(* IEC 61131-3 sources: Lua/, 14 files *)

(* ---- 1#真空脱水.st ---- *)
FUNCTION_BLOCK Dewater
    VAR_STATIC
        // 1#真空脱水控制流--结构体
        TYPE Dewater_1: STRUCT
                bnt_run: BOOL; (* 启动按钮 *)
                bnt_stop: BOOL; (* 停止按钮 *)
                bnt_manual: BOOL; (* 手动按钮 *)
                state: INT; (* 状态 *)
                error_id: INT; (* 错误 *)
                TYPE run: STRUCT
                        todo: BOOL; (* 初始化 *)
                        busy: BOOL; (* 执行中 *)
                        STEP: INT; (* 步数 *)
                        in_time: WORD; (* 计时器输入IN *)
                        skip: BOOL; (* 跳过 *)
                    END_STRUCT
                END_TYPE
                TYPE stop: STRUCT
                        todo: BOOL; (* 初始化 *)
                        busy: BOOL; (* 执行中 *)
                        STEP: INT; (* 步数 *)
                        in_time: WORD; (* 计时器输入IN *)
                        skip: BOOL; (* 跳过 *)
                    END_STRUCT
                END_TYPE
            END_STRUCT
        END_TYPE
        // 1#真空脱水设置时间--结构体
        TYPE Retain_time_D_1 : STRUCT
                preTime : DINT; (* 预处理时间 *)
                openTime_1 : DINT; (* 真空脱水时间 *)
                openTime_2 : DINT; (* 真空脱水时间 *)
                delayTime : DINT; (* 延迟时间 *)
                loopTime : DINT; (* 循环时间 *)
            END_STRUCT
        END_TYPE
        // 1#真空脱水计时器--数组
        Timer_D_1 : ARRAY [0..3] OF TON_TIME;

        CIP_1: "CIP"
        bnt_run: BOOL			启动按钮
        bnt_stop: BOOL			停止按钮
        todo: BOOL			    初始化
        busy: BOOL			    执行中
        step: INT			    步数
        in_time: WORD			计时器输入IN
        error: INT			    错误
        state: INT			    状态

	    Timer_CIP_1	Array[0..10] of TON_TIME

        Retain_time_CIP_1: "CIP_time"
        preTime: DINT
        stepTime_1: DINT
        stepTime_2: DINT
        T102: DINT
        T103: DINT
        T104: DINT
        T105: DINT
        T106: DINT
        T110: DINT
        T107: DINT
        T108: DINT
        T109: DINT
    END_VAR

    /*
        真空脱水一键启动
    */
    // 计时器
    Timer_D_1[0] (IN := #Dewater_1.run.in_time.%X0, PT := #Retain_time_D_1.preTime);
    Timer_D_1[1] (IN := #Dewater_1.run.in_time.%X1, PT := #Retain_time_D_1.openTime_1);

    // 预处理
    IF "Global".Emergency.Dewater_1 THEN
        IF #Dewater_1.bnt_run AND NOT #Dewater_1.run.busy THEN
            "V8016-O" := FALSE;
            "V8021-O" := FALSE;
            "V8011-O" := FALSE;
            "V8026-O" := TRUE;
            #Dewater_1.run.todo := TRUE;
        END_IF;
        IF #Dewater_1.run.todo THEN
            #Dewater_1.state := 1;
            #Dewater_1.run.step := 1;
            #Dewater_1.run.skip := FALSE;
            #Dewater_1.run.in_time := 0;
            #Dewater_1.run.in_time.%X0 := TRUE;
            "ALARM3-O" := TRUE;
            #Dewater_1.bnt_run := FALSE;
        END_IF;
        IF #Dewater_1.run.in_time.%X0 AND #Timer_D_1[0].Q THEN
            #Dewater_1.run.busy := TRUE;
            #Dewater_1.run.todo := FALSE;
            "ALARM3-O" := FALSE;
        ELSE
            #Dewater_1.run.busy := FALSE;
        END_IF;
    ELSE
        #Dewater_1.state := 0;
        #Dewater_1.run.step := 0;
        #Dewater_1.run.in_time := 0;
        #Dewater_1.stop.step := 0;
        #Dewater_1.stop.in_time := 0;
        "ALARM3-O" := FALSE;
    END_IF;

    // 手动时
    IF "Global".Emergency.Dewater_1 AND #Dewater_1.bnt_manual THEN
        #Dewater_1.state := 2;
        #Dewater_1.run.step := 0;
        #Dewater_1.run.in_time := 0;
        #Dewater_1.stop.step := 0;
        #Dewater_1.stop.in_time := 0;
    END_IF;

    // 停止时
    IF "Global".Emergency.Dewater_1 AND #Dewater_1.bnt_stop THEN
        #Dewater_1.state := 3;
        #Dewater_1.run.step := 0;
        #Dewater_1.run.in_time := 0;
    END_IF;

    // 启动中
    IF #Dewater_1.run.busy AND Dewater_1.state = 1 THEN
        // 第1步
        IF #Dewater_1.run.step = 1 THEN
            IF NOT "KV7001-O" THEN
                "KV7001-O" := TRUE;
                #Dewater_1.run.step := 2;
                RETURN;
            END_IF;
            IF "KV7001-O" THEN
                #Dewater_1.run.skip := TRUE;
                #Dewater_1.run.step := 2;
            END_IF;
        END_IF;
        // 第2步
        IF #Dewater_1.run.step = 2 THEN
            IF NOT "A7001-DO" THEN
                IF #Dewater_1.run.skip THEN
                    "A7001-DO" := TRUE;
                    #Dewater_1.run.skip := FALSE;
                    #Dewater_1.run.step := 3;
                    RETURN;
                END_IF;
                #Dewater_1.run.in_time.%X1 := TRUE;
                IF #Dewater_1.run.in_time.%X1 AND #Timer_D_1[1].Q THEN
                    "A7001-DO" := TRUE;
                    #Dewater_1.run.in_time.%X1 := FALSE;
                    #Dewater_1.run.step := 3;
                    RETURN;
                END_IF;
            END_IF;
            IF "A7001-DO" THEN
                #Dewater_1.run.step := 3;
            END_IF;
        END_IF;
        // 第3步
        IF #Dewater_1.run.step = 3 THEN
            IF NOT "F7001-DO" THEN
                IF #Dewater_1.run.skip THEN
                    "F7001-DO" := TRUE;
                    #Dewater_1.run.skip := FALSE;
                    #Dewater_1.run.step := 4;
                    RETURN;
                END_IF;
                #Dewater_1.run.in_time.%X1 := TRUE;
                IF #Dewater_1.run.in_time.%X1 AND #Timer_D_1[1].Q THEN
                    "F7001-DO" := TRUE;
                    #Dewater_1.run.in_time.%X1 := FALSE;
                    #Dewater_1.run.step := 4;
                    RETURN;
                END_IF;
            END_IF;
            IF "F7001-DO" THEN
                #Dewater_1.run.step := 4;
            END_IF;
        END_IF;
        // 第4步
        IF #Dewater_1.run.step = 4 THEN
            IF NOT ( "V8001-O" AND NOT "V8006-O" ) THEN
                IF #Dewater_1.run.skip THEN
                    "V8001-O" := TRUE;
                    "V8006-O" := FALSE;
                    #Dewater_1.run.skip := FALSE;
                    #Dewater_1.run.step := 5;
                    RETURN;
                END_IF;
                #Dewater_1.run.in_time.%X1 := TRUE;
                IF #Dewater_1.run.in_time.%X1 AND #Timer_D_1[1].Q THEN
                    "V8001-O" := TRUE;
                    "V8006-O" := FALSE;
                    #Dewater_1.run.in_time.%X1 := FALSE;
                    #Dewater_1.run.step := 5;
                    RETURN;
                END_IF;
            END_IF;
            IF "V8001-O" AND NOT "V8006-O" THEN
                #Dewater_1.run.step := 5;
            END_IF;
        END_IF;
        // 第5步
        IF #Dewater_1.run.step = 5 THEN
            IF NOT "P8001-DO" THEN
                IF #Dewater_1.run.skip THEN
                    "P8001-DO" := TRUE;
                    #Dewater_1.run.skip := FALSE;
                    #Dewater_1.run.step := 6;
                    RETURN;
                END_IF;
                #Dewater_1.run.in_time.%X1 := TRUE;
                IF #Dewater_1.run.in_time.%X1 AND #Timer_D_1[1].Q THEN
                    "P8001-DO" := TRUE;
                    #Dewater_1.run.in_time.%X1 := FALSE;
                    #Dewater_1.run.step := 6;
                    RETURN;
                END_IF;
            END_IF;
            IF "P8001-DO" THEN
                #Dewater_1.run.step := 6;
            END_IF;
        END_IF;
        // 第6步
        IF #Dewater_1.run.step = 6 THEN
            IF NOT "T7001-DO" THEN
                IF #Dewater_1.run.skip THEN
                    "T7001-DO" := TRUE;
                    #Dewater_1.run.skip := FALSE;
                    #Dewater_1.run.step := 7;
                    RETURN;
                END_IF;
                #Dewater_1.run.in_time.%X1 := TRUE;
                IF #Dewater_1.run.in_time.%X1 AND #Timer_D_1[1].Q THEN
                    "T7001-DO" := TRUE;
                    #Dewater_1.run.in_time.%X1 := FALSE;
                    #Dewater_1.run.step := 7;
                    RETURN;
                END_IF;
            END_IF;
            IF "T7001-DO" THEN
                #Dewater_1.run.step := 7;
            END_IF;
        END_IF;
        // 第7步
        IF #Dewater_1.run.step = 7 THEN
            IF NOT "P7006-DO" THEN
                IF #Dewater_1.run.skip THEN
                    IF "Global".Disp_LIT_7001 > "Global".set_LIT_7001 THEN
                        "P7006-DO" := TRUE;
                        #Dewater_1.run.skip := FALSE;
                        #Dewater_1.run.step := 8;
                        RETURN;
                    ELSE
                        RETURN;
                    END_IF;
                END_IF;
                IF "Global".Disp_LIT_7001 > "Global".set_LIT_7001 THEN
                    #Dewater_1.run.in_time.%X1 := TRUE;
                    IF #Dewater_1.run.in_time.%X1 AND #Timer_D_1[1].Q THEN
                        "P7006-DO" := TRUE;
                        #Dewater_1.run.in_time.%X1 := FALSE;
                        #Dewater_1.run.step := 8;
                        RETURN;
                    END_IF;
                END_IF;
            END_IF;
            IF "P7006-DO" THEN
                #Dewater_1.run.step := 8;
            END_IF;
        END_IF
        // 第8步
        IF #Dewater_1.run.step = 8 THEN
            IF NOT "V7001-O" THEN
                IF #Dewater_1.run.skip THEN
                    "V7001-O" := TRUE;
                    #Dewater_1.run.skip := FALSE;
                    #Dewater_1.run.step := 9;
                    RETURN;
                END_IF;
                #Dewater_1.run.in_time.%X1 := TRUE;
                IF #Dewater_1.run.in_time.%X1 AND #Timer_D_1[1].Q THEN
                    "V7001-O" := TRUE;
                    #Dewater_1.run.in_time.%X1 := FALSE;
                    #Dewater_1.run.step := 9;
                    RETURN;
                END_IF;
            END_IF;
            IF "V7001-O" THEN
                #Dewater_1.run.step := 9;
            END_IF;
        END_IF;
        // 第9步
        IF #Dewater_1.run.step = 9 THEN
            IF NOT "P7001-DO" THEN
                #Dewater_1.run.in_time.%X1 := TRUE;
                IF #Dewater_1.run.in_time.%X1 AND #Timer_D_1[1].Q THEN
                    "P7001-DO" := TRUE;
                    #Dewater_1.run.in_time := 0;
                    #Dewater_1.run.step := 100;
                    RETURN;
                END_IF;
            END_IF;
            IF "P7001-DO" THEN
                #Dewater_1.run.in_time := 0;
                #Dewater_1.run.step := 100;
            END_IF;
        END_IF;
    END_IF;

    /*
        CIP在线清洗
    */
    REGION 计时器
        #Timer_CIP_1[0](IN:=#CIP_1.in_time.%X0, PT:=#Retain_time_CIP_1.preTime);
        #Timer_CIP_1[1](IN := #CIP_1.in_time.%X1, PT := #Retain_time_CIP_1.stepTime_1);
        #Timer_CIP_1[2](IN := #CIP_1.in_time.%X2, PT := #Retain_time_CIP_1.T102);
        #Timer_CIP_1[3](IN := #CIP_1.in_time.%X3, PT := #Retain_time_CIP_1.T103);
        #Timer_CIP_1[4](IN := #CIP_1.in_time.%X4, PT := #Retain_time_CIP_1.T104);
        #Timer_CIP_1[5](IN := #CIP_1.in_time.%X5, PT := #Retain_time_CIP_1.T105);
        #Timer_CIP_1[6](IN := #CIP_1.in_time.%X6, PT := #Retain_time_CIP_1.T106);
        #Timer_CIP_1[7](IN := #CIP_1.in_time.%X7, PT := #Retain_time_CIP_1.T107);
        #Timer_CIP_1[8](IN := #CIP_1.in_time.%X8, PT := #Retain_time_CIP_1.T108);
        #Timer_CIP_1[9](IN := #CIP_1.in_time.%X9, PT := #Retain_time_CIP_1.T109);
        #Timer_CIP_1[10](IN := #CIP_1.in_time.%X10, PT := #Retain_time_CIP_1.T110);
    END_REGION

    REGION 预处理
        // 初始化
        IF "Global".Emergency.Dewater_1 THEN
            IF #Dewater_1.state = 1 AND #Dewater_1.run.step = 100 AND #CIP_1.bnt_run AND NOT #CIP_1.busy THEN
                #CIP_1.todo := TRUE;
            END_IF;
            IF #CIP_1.todo THEN
                #CIP_1.state := 1;
                #CIP_1.step := 1;
                #CIP_1.in_time := 0;
                #CIP_1.in_time.%X0 := TRUE;
                #CIP_1.bnt_run := FALSE;
                #CIP_1.todo := FALSE;
            END_IF;
            IF #CIP_1.in_time.%X0 AND #Timer_CIP_1[0].Q THEN
                #CIP_1.busy := TRUE;
            ELSE
                #CIP_1.busy := FALSE;
            END_IF;
        ELSE
            #CIP_1.state := 0;
            #CIP_1.step := 0;
            #CIP_1.in_time := 0;
        END_IF;
    END_REGION

    REGION CIP运行中
        IF #CIP_1.busy AND #CIP_1.state = 1 THEN
            // step 1
            IF #CIP_1.step = 1 THEN
                "V8006-O" := TRUE;
                #CIP_1.step := 2;
            END_IF;
            // step 2
            IF #CIP_1.step = 2 THEN
                #CIP_1.in_time.%X2 := TRUE;
                IF #CIP_1.in_time.%X2 AND #Timer_CIP_1[2].Q THEN
                    "V8001-O" := FALSE;
                    #CIP_1.in_time.%X2:= FALSE;
                    #CIP_1.step := 3;
                END_IF;
            END_IF;
            // step 3
            IF #CIP_1.step = 3 THEN
                #CIP_1.in_time.%X3 := TRUE;
                IF #CIP_1.in_time.%X3 AND #Timer_CIP_1[3].Q THEN
                    "P8001-DO" := FALSE;
                    "Global".PID_7101.Man_enable := TRUE;
                    "Global".PID_7101.Man_value := 0;
                    "V8006-O" := FALSE;
                    "V8011-O" := TRUE;
                    #CIP_1.in_time.%X3 := FALSE;
                    #CIP_1.step := 4;
                END_IF;
            END_IF;
            // step 4
            IF #CIP_1.step = 4 THEN
                #CIP_1.in_time.%X4 := TRUE;
                IF #CIP_1.in_time.%X4 AND #Timer_CIP_1[4].Q THEN
                    "V8011-O" := FALSE;
                    #CIP_1.in_time.%X4 := FALSE;
                    #CIP_1.step := 5;
                END_IF;
            END_IF;
            // step 5
            IF #CIP_1.step = 5 THEN
                #CIP_1.in_time.%X1 := TRUE;
                IF #CIP_1.in_time.%X1 AND #Timer_CIP_1[1].Q THEN
                    "KV7001-O" := FALSE;
                    #CIP_1.in_time.%X1 := FALSE;
                    #CIP_1.step := 6;
                    RETURN;
                END_IF;
            END_IF;
            // step 6
            IF #CIP_1.step = 6 THEN
                #CIP_1.in_time.%X1 := TRUE;
                IF #CIP_1.in_time.%X1 AND #Timer_CIP_1[1].Q THEN
                    "P7001-DO" := FALSE;
                    "V7001-O" := FALSE;
                    #CIP_1.in_time.%X1 := FALSE;
                    #CIP_1.step := 7;
                    RETURN;
                END_IF;
            END_IF;
            // step 7
            IF #CIP_1.step = 7 THEN
                #CIP_1.in_time.%X1 := TRUE;
                IF #CIP_1.in_time.%X1 AND #Timer_CIP_1[1].Q THEN
                    "P7006-DO" := FALSE;
                    #CIP_1.in_time.%X1 := FALSE;
                    #CIP_1.step := 8;
                    RETURN;
                END_IF;
            END_IF;
            // step 8
            IF #CIP_1.step = 8 THEN
                #CIP_1.in_time.%X1 := TRUE;
                IF #CIP_1.in_time.%X1 AND #Timer_CIP_1[1].Q THEN
                    "T7001-DO" := FALSE;
                    #CIP_1.in_time.%X1 := FALSE;
                    #CIP_1.step := 9;
                    RETURN;
                END_IF;
            END_IF;
            // step 9
            IF #CIP_1.step = 9 THEN
                #CIP_1.in_time.%X1 := TRUE;
                IF #CIP_1.in_time.%X1 AND #Timer_CIP_1[1].Q THEN
                    "V8016-O" := TRUE;
                    "V8017-O" := FALSE;
                    "V8018-O" := FALSE;
                    "V8019-O" := FALSE;
                    "V8020-O" := FALSE;
                    "V8021-O" := FALSE;
                    #CIP_1.in_time.%X1 := FALSE;
                    #CIP_1.step := 901;
                    RETURN;
                END_IF;
            END_IF;
            // step 901
            IF #CIP_1.step = 901 THEN
                #CIP_1.in_time.%X1 := TRUE;
                IF #CIP_1.in_time.%X1 AND #Timer_CIP_1[1].Q THEN
                    "P8007-DO" := TRUE;
                    #CIP_1.in_time.%X1 := FALSE;
                    #CIP_1.step := 10;
                    RETURN;
                END_IF;
            END_IF;
            // step 10
            IF #CIP_1.step = 10 THEN
                #CIP_1.in_time.%X5 := TRUE;
                IF #CIP_1.in_time.%X5 AND #Timer_CIP_1[5].Q THEN
                    "P8007-DO" := FALSE;
                    "V8016-O" := FALSE;
                    #CIP_1.in_time.%X5 := FALSE;
                    #CIP_1.step := 11;
                END_IF;
            END_IF;
            // step 11
            IF #CIP_1.step = 11 THEN
                #CIP_1.in_time.%X6 := TRUE;
                IF #CIP_1.in_time.%X6 AND #Timer_CIP_1[6].Q THEN
                    "V8026-O" := TRUE;
                    "V8032-O" := TRUE;
                    #CIP_1.in_time.%X6 := FALSE;
                    #CIP_1.step := 12;
                END_IF;
            END_IF;
            // step 12
            IF #CIP_1.step = 12 THEN
                #CIP_1.in_time.%X10 := TRUE;
                IF #CIP_1.in_time.%X10 AND #Timer_CIP_1[10].Q THEN
                    "V8032-O" := FALSE;
                    "Global".set_Hz_F7001 := 10.0;
                    #CIP_1.in_time.%X10 := FALSE;
                    #CIP_1.step := 13;
                END_IF;
            END_IF;
            // step 13
            IF #CIP_1.step = 13 THEN
                #CIP_1.in_time.%X1 := TRUE;
                IF #CIP_1.in_time.%X1 AND #Timer_CIP_1[1].Q THEN
                    "V8016-O" := TRUE;
                    "V8017-O" := FALSE;
                    "V8018-O" := FALSE;
                    "V8019-O" := FALSE;
                    "V8020-O" := FALSE;
                    "V8021-O" := FALSE;
                    #CIP_1.in_time.%X1 := FALSE;
                    #CIP_1.step := 1301;
                    RETURN;
                END_IF;
            END_IF;
            // step 1301
            IF #CIP_1.step = 1301 THEN
                #CIP_1.in_time.%X1 := TRUE;
                IF #CIP_1.in_time.%X1 AND #Timer_CIP_1[1].Q THEN
                    "P8007-DO" := TRUE;
                    #CIP_1.in_time.%X1 := FALSE;
                    #CIP_1.step := 14;
                    RETURN;
                END_IF;
            END_IF;
            // step 14
            IF #CIP_1.step = 14 THEN
                #CIP_1.in_time.%X7 := TRUE;
                IF #CIP_1.in_time.%X7 AND #Timer_CIP_1[7].Q THEN
                    "P8007-DO" := FALSE;
                    "V8016-O" := FALSE;
                    #CIP_1.in_time.%X7 := FALSE;
                    #CIP_1.step := 15;
                END_IF;
            END_IF;
            // step 15
            IF #CIP_1.step = 15 THEN
                #CIP_1.in_time.%X8 := TRUE;
                IF #CIP_1.in_time.%X8 AND #Timer_CIP_1[8].Q THEN
                    "V8026-O" := FALSE;
                    "V8031-O" := TRUE;
                    #CIP_1.in_time.%X8 := FALSE;
                    #CIP_1.step := 16;
                END_IF;
            END_IF;
            // step 16
            IF #CIP_1.step = 16 THEN
                #CIP_1.in_time.%X9 := TRUE;
                IF #CIP_1.in_time.%X9 AND #Timer_CIP_1[9].Q THEN
                    "V8031-O" := FALSE;
                    #CIP_1.in_time.%X9 := FALSE;
                    #CIP_1.step := 17;
                END_IF;
            END_IF;
            // step 17
            IF #CIP_1.step = 17 THEN
                #CIP_1.in_time.%X1 := TRUE;
                IF #CIP_1.in_time.%X1 AND #Timer_CIP_1[1].Q THEN
                    "A7001-DO" := FALSE;
                    #CIP_1.in_time.%X1 := FALSE;
                    #CIP_1.step := 18;
                    RETURN;
                END_IF;
            END_IF;
            // step 18
            IF #CIP_1.step = 18 THEN
                #CIP_1.in_time.%X1 := TRUE;
                IF #CIP_1.in_time.%X1 AND #Timer_CIP_1[1].Q THEN
                    "F7001-DO" := FALSE;
                    #CIP_1.in_time.%X1 := FALSE;
                    #CIP_1.step := 19;
                END_IF;
            END_IF;
        END_IF;
    END_REGION
END_FUNCTION_BLOCK

(* ---- 真空脱水_3_25.st ---- *)
FUNCTION_BLOCK Dewater
    VAR_STAT
        // 1#真空脱水控制流--结构体
        TYPE Dewater_1: STRUCT
                bnt_run: BOOL; (* 启动按钮 *)
                bnt_stop: BOOL; (* 停止按钮 *)
                bnt_manual: BOOL; (* 手动按钮 *)
                state: INT; (* 状态 *)
                TYPE run: STRUCT
                        todo: BOOL; (* 初始化 *)
                        busy: BOOL; (* 执行中 *)
                        STEP: INT; (* 步数 *)
                        in_time: WORD; (* 计时器输入IN *)
                        skip: BOOL; (* 跳过 *)
                    END_STRUCT
                END_TYPE
                TYPE stop: STRUCT
                        todo: BOOL; (* 初始化 *)
                        busy: BOOL; (* 执行中 *)
                        STEP: INT; (* 步数 *)
                        in_time: WORD; (* 计时器输入IN *)
                        skip: BOOL; (* 跳过 *)
                    END_STRUCT
                END_TYPE
            END_STRUCT
        END_TYPE
        // 1#真空脱水设置时间--结构体
        TYPE Retain_time_D_1 : STRUCT
                preTime : DINT; (* 预处理时间 *)
                openTime_1 : DINT; (* 真空脱水时间 *)
                openTime_2 : DINT; (* 真空脱水时间 *)
                delayTime : DINT; (* 延迟时间 *)
                loopTime : DINT; (* 循环时间 *)
            END_STRUCT
        END_TYPE
        // 1#真空脱水计时器--数组
        Timer_D_1 : ARRAY [0..3] OF TON_TIME;
    END_VAR

    // 计时器
    Timer_D_1[0](IN := #Dewater_1.run.in_time.%X0, PT := #Retain_time_D_1.preTime);
    Timer_D_1[1](IN := #Dewater_1.run.in_time.%X0, PT := #Retain_time_D_1.openTime_1);

    // 预处理
    IF "Global".Emergency.Dewater_1 THEN
    IF #Dewater_1.bnt_run AND NOT #Dewater_1.run.busy THEN
        #Dewater_1.run.todo := TRUE;
    END_IF;
    IF #Dewater_1.run.todo THEN
        #Dewater_1.state := 1;
        #Dewater_1.run.step := 1;
        #Dewater_1.run.skip := FALSE;
        #Dewater_1.run.in_time := 0;
        #Dewater_1.run.in_time.%X0 := TRUE;
        "ALARM1-O" := TRUE;
        #Dewater_1.bnt_run := FALSE;
        #Dewater_1.run.todo := FALSE;
    END_IF;

    END_IF;

END_FUNCTION_BLOCK

(* ---- 顺序启动_最新.st ---- *)
FUNCTION_BLOCK Extraction
    VAR_GLOBAL
        //提取单元自动启动关键属性--结构体
        TYPE Common_M_1_run : STRUCT
                bnt_run : BOOL; (* 自动启动 *)
                bnt_stop : BOOL; (* 自动停止 *)
                todo : BOOL; (* 是否跳过步骤1 *)
                busy : BOOL; (* 自动正在执行 *)
                step : INT; (* 自动运行步骤 *)
                in_time : WORD; (* 控制计时器输入IN通断 *)
                manual_enable : BOOL; (* 手动模式按钮 *)
                state : INT; (* 提取单元状态都在此处显示 *)
            END_STRUCT
        END_TYPE

        //提取单元自动启动设定时间--结构体
        TYPE Retain_M5000_run : STRUCT
                preTime : DINT; (* 自动启动预处理时间 *)
                openTime_1 : DINT; (* 自动启动电机延时打开时间 *)
            END_STRUCT
        END_TYPE

        //提取单元启动--通电延时计时器
        Timer_M5000_run : ARRAY[0..2] of TON_TIME;
        (*
            Timer_M5000_run[0]......预处理--计时器
            Timer_M5000_run[1]......电机打开延时--计时器
        *)
    END_VAR

    /* *
    **计时器
    */
    #Timer_M5000_run[0](IN := #Common_M_1_run.in_time.%X0, PT := #Retain_M5000_run.preTime);
    #Timer_M5000_run[1](IN := #Common_M_1_run.in_time.%X1, PT := #Retain_M5000_run.openTime_1);

    /* *
    **预处理
    */
    IF "Global".Emergency.Extraction_1 AND #Common_M_1_run.bnt_run AND NOT #Common_M_1_run.busy THEN
    #Common_M_1_run.state := 1;
    #Common_M_1_run.step := 1;
    #Common_M_1_run.in_time := 0;
    #Common_M_1_run.todo := FALSE;
    #Common_M_1_run.in_time.%X0 := TRUE;
    END_IF;
    IF #Common_M_1_run.in_time.%X0 AND #Timer_M5000_run[0].Q THEN
    #Common_M_1_run.bnt_run := FALSE;
    #Common_M_1_run.busy := TRUE;
    ELSE
    #Common_M_1_run.busy := FALSE;
    END_IF;

    //急停时
    IF NOT "Global".Emergency.Extraction_1 THEN
    #Common_M_1_run.state := 0;
    #Common_M_1_run.step := 0;
    #Common_M_1_run.in_time := 0;
    #Common_M_1_run.bnt_run := FALSE;
    END_IF;

    //手动时
    IF "Global".Emergency.Extraction_1 AND #Common_M_1_run.manual_enable THEN
    #Common_M_1_run.state := 2;
    #Common_M_1_run.step := 0;
    #Common_M_1_run.in_time := 0;
    #Common_M_1_run.bnt_run := FALSE;
    END_IF;

    //停止时
    IF "Global".Emergency.Extraction_1 AND #Common_M_1_run.bnt_stop THEN
    #Common_M_1_run.step := 0;
    #Common_M_1_run.in_time := 0;
    #Common_M_1_run.bnt_run := FALSE;
    END_IF;

    /* *
    **运行时
    */
    IF #Common_M_1_run.busy AND #Common_M_1_run.state = 1 THEN
    //step1
    IF #Common_M_1_run.step = 1 THEN
        IF NOT "M5203-DO" THEN
            "M5203-DO" := TRUE;
            #Common_M_1_run.step := 2;
            RETURN;
        END_IF;
        IF "M5203-DO" THEN
            #Common_M_1_run.todo := TRUE;
            #Common_M_1_run.step := 2;
        END_IF;
    END_IF;
    //step2
    IF #Common_M_1_run.step = 2 THEN
        IF NOT "M5103-DO" THEN
            IF #Common_M_1_run.todo THEN
                "M5103-DO" := TRUE;
                #Common_M_1_run.todo := FALSE;
                #Common_M_1_run.step := 3;
                RETURN;
            END_IF;
            #Common_M_1_run.in_time.%X1 := TRUE;
            IF #Common_M_1_run.in_time.%X1 AND #Timer_M5000_run[1].Q THEN
                "M5103-DO" := TRUE;
                #Common_M_1_run.in_time.%X1 := FALSE;
                #Common_M_1_run.step := 3;
                RETURN;
            END_IF;
        END_IF;
        IF "M5103-DO" THEN
            #Common_M_1_run.step := 3;
        END_IF;
    END_IF;
    //step3
    IF #Common_M_1_run.step = 3 THEN
        IF NOT "M5202-DO" THEN
            IF #Common_M_1_run.todo THEN
                "M5202-DO" := TRUE;
                #Common_M_1_run.todo := FALSE;
                #Common_M_1_run.step := 4;
                RETURN;
            END_IF;
            #Common_M_1_run.in_time.%X1 := TRUE;
            IF #Common_M_1_run.in_time.%X1 AND #Timer_M5000_run[1].Q THEN
                "M5202-DO" := TRUE;
                #Common_M_1_run.in_time.%X1 := FALSE;
                #Common_M_1_run.step := 4;
                RETURN;
            END_IF;
        END_IF;
        IF "M5202-DO" THEN
            #Common_M_1_run.step := 4;
        END_IF;
    END_IF;
    //step4
    IF #Common_M_1_run.step = 4 THEN
        IF NOT "M5102-DO" THEN
            IF #Common_M_1_run.todo THEN
                "M5102-DO" := TRUE;
                #Common_M_1_run.todo := FALSE;
                #Common_M_1_run.step := 5;
                RETURN;
            END_IF;
            #Common_M_1_run.in_time.%X1 := TRUE;
            IF #Common_M_1_run.in_time.%X1 AND #Timer_M5000_run[1].Q THEN
                "M5102-DO" := TRUE;
                #Common_M_1_run.in_time.%X1 := FALSE;
                #Common_M_1_run.step := 5;
                RETURN;
            END_IF;
        END_IF;
        IF "M5102-DO" THEN
            #Common_M_1_run.step := 5;
        END_IF;
    END_IF;
    //step5
    IF #Common_M_1_run.step = 5 THEN
        IF NOT "M5401-DO" THEN
            IF #Common_M_1_run.todo THEN
                "M5401-DO" := TRUE;
                #Common_M_1_run.todo := FALSE;
                #Common_M_1_run.step := 6;
                RETURN;
            END_IF;
            #Common_M_1_run.in_time.%X1 := TRUE;
            IF #Common_M_1_run.in_time.%X1 AND #Timer_M5000_run[1].Q THEN
                "M5401-DO" := TRUE;
                #Common_M_1_run.in_time.%X1 := FALSE;
                #Common_M_1_run.step := 6;
                RETURN;
            END_IF;
        END_IF;
        IF "M5401-DO" THEN
            #Common_M_1_run.step := 6;
        END_IF;
    END_IF;
    //step6
    IF #Common_M_1_run.step = 6 THEN
        IF NOT "M5301-DO" THEN
            IF #Common_M_1_run.todo THEN
                "M5301-DO" := TRUE;
                #Common_M_1_run.todo := FALSE;
                #Common_M_1_run.step := 7;
                RETURN;
            END_IF;
            #Common_M_1_run.in_time.%X1 := TRUE;
            IF #Common_M_1_run.in_time.%X1 AND #Timer_M5000_run[1].Q THEN
                "M5301-DO" := TRUE;
                #Common_M_1_run.in_time.%X1 := FALSE;
                #Common_M_1_run.step := 7;
                RETURN;
            END_IF;
        END_IF;
        IF "M5301-DO" THEN
            #Common_M_1_run.step := 7;
        END_IF;
    END_IF;
    //step7
    IF #Common_M_1_run.step = 7 THEN
        IF NOT "M5201-DO" THEN
            IF #Common_M_1_run.todo THEN
                "M5201-DO" := TRUE;
                #Common_M_1_run.todo := FALSE;
                #Common_M_1_run.step := 8;
                RETURN;
            END_IF;
            #Common_M_1_run.in_time.%X1 := TRUE;
            IF #Common_M_1_run.in_time.%X1 AND #Timer_M5000_run[1].Q THEN
                "M5201-DO" := TRUE;
                #Common_M_1_run.in_time.%X1 := FALSE;
                #Common_M_1_run.step := 8;
                RETURN;
            END_IF;
        END_IF;
        IF "M5201-DO" THEN
            #Common_M_1_run.step := 8;
        END_IF;
    END_IF;
    //step8
    IF #Common_M_1_run.step = 8 THEN
        IF NOT "M5101-DO" THEN
            IF #Common_M_1_run.todo THEN
                "M5101-DO" := TRUE;
                #Common_M_1_run.todo := FALSE;
                #Common_M_1_run.step := 9;
                RETURN;
            END_IF;
            #Common_M_1_run.in_time.%X1 := TRUE;
            IF #Common_M_1_run.in_time.%X1 AND #Timer_M5000_run[1].Q THEN
                "M5101-DO" := TRUE;
                #Common_M_1_run.in_time.%X1 := FALSE;
                #Common_M_1_run.step := 9;
                RETURN;
            END_IF;
        END_IF;
        IF "M5101-DO" THEN
            #Common_M_1_run.step := 9;
        END_IF;
    END_IF;
    //step9
    IF #Common_M_1_run.step = 9 THEN
        IF NOT "P5005-DO" THEN
            IF #Common_M_1_run.todo THEN
                "P5005-DO" := TRUE;
                #Common_M_1_run.todo := FALSE;
                #Common_M_1_run.step := 10;
                RETURN;
            END_IF;
            #Common_M_1_run.in_time.%X1 := TRUE;
            IF #Common_M_1_run.in_time.%X1 AND #Timer_M5000_run[1].Q THEN
                "P5005-DO" := TRUE;
                #Common_M_1_run.in_time.%X1 := FALSE;
                #Common_M_1_run.step := 10;
                RETURN;
            END_IF;
        END_IF;
        IF "P5005-DO" THEN
            #Common_M_1_run.step := 10;
        END_IF;
    END_IF;
    //step10
    IF #Common_M_1_run.step = 10 THEN
        IF NOT "P5003-DO" THEN
            IF #Common_M_1_run.todo THEN
                "P5003-DO" := TRUE;
                #Common_M_1_run.todo := FALSE;
                #Common_M_1_run.step := 11;
                RETURN;
            END_IF;
            #Common_M_1_run.in_time.%X1 := TRUE;
            IF #Common_M_1_run.in_time.%X1 AND #Timer_M5000_run[1].Q THEN
                "P5003-DO" := TRUE;
                #Common_M_1_run.in_time.%X1 := FALSE;
                #Common_M_1_run.step := 11;
                RETURN;
            END_IF;
        END_IF;
        IF "P5003-DO" THEN
            #Common_M_1_run.step := 11;
        END_IF;
    END_IF;
    //step11
    IF #Common_M_1_run.step = 11 THEN
        IF NOT "P5201-DO" THEN
            IF #Common_M_1_run.todo THEN
                "P5201-DO" := TRUE;
                #Common_M_1_run.todo := FALSE;
                #Common_M_1_run.step := 12;
                RETURN;
            END_IF;
            #Common_M_1_run.in_time.%X1 := TRUE;
            IF #Common_M_1_run.in_time.%X1 AND #Timer_M5000_run[1].Q THEN
                "P5201-DO" := TRUE;
                #Common_M_1_run.in_time.%X1 := FALSE;
                #Common_M_1_run.step := 12;
                RETURN;
            END_IF;
        END_IF;
        IF "P5201-DO" THEN
            #Common_M_1_run.step := 12;
        END_IF;
    END_IF;
    //step12
    IF #Common_M_1_run.step = 12 THEN
        IF NOT "P5101-DO" THEN
            IF #Common_M_1_run.todo THEN
                "P5101-DO" := TRUE;
                #Common_M_1_run.todo := FALSE;
                #Common_M_1_run.step := 13;
                RETURN;
            END_IF;
            #Common_M_1_run.in_time.%X1 := TRUE;
            IF #Common_M_1_run.in_time.%X1 AND #Timer_M5000_run[1].Q THEN
                "P5101-DO" := TRUE;
                #Common_M_1_run.in_time.%X1 := FALSE;
                #Common_M_1_run.step := 13;
                RETURN;
            END_IF;
        END_IF;
        IF "P5101-DO" THEN
            #Common_M_1_run.step := 13;
        END_IF;
    END_IF;
    //step13
    IF #Common_M_1_run.step = 13 THEN
        IF NOT "P5206-DO" THEN
            IF #Common_M_1_run.todo THEN
                "P5206-DO" := TRUE;
                #Common_M_1_run.todo := FALSE;
                #Common_M_1_run.step := 14;
                RETURN;
            END_IF;
            #Common_M_1_run.in_time.%X1 := TRUE;
            IF #Common_M_1_run.in_time.%X1 AND #Timer_M5000_run[1].Q THEN
                "P5206-DO" := TRUE;
                #Common_M_1_run.in_time.%X1 := FALSE;
                #Common_M_1_run.step := 14;
                RETURN;
            END_IF;
        END_IF;
        IF "P5206-DO" THEN
            #Common_M_1_run.step := 14;
        END_IF;
    END_IF;
    //step14
    IF #Common_M_1_run.step = 14 THEN
        IF NOT "P5106-DO" THEN
            IF #Common_M_1_run.todo THEN
                "P5106-DO" := TRUE;
                #Common_M_1_run.todo := FALSE;
                #Common_M_1_run.step := 15;
                RETURN;
            END_IF;
            #Common_M_1_run.in_time.%X1 := TRUE;
            IF #Common_M_1_run.in_time.%X1 AND #Timer_M5000_run[1].Q THEN
                "P5106-DO" := TRUE;
                #Common_M_1_run.in_time.%X1 := FALSE;
                #Common_M_1_run.step := 15;
                RETURN;
            END_IF;
        END_IF;
        IF "P5106-DO" THEN
            #Common_M_1_run.step := 15;
        END_IF;
    END_IF;
    //step15
    IF #Common_M_1_run.step = 15 THEN
        IF NOT "P5204-DO" THEN
            IF #Common_M_1_run.todo THEN
                "P5204-DO" := TRUE;
                #Common_M_1_run.todo := FALSE;
                #Common_M_1_run.step := 16;
                RETURN;
            END_IF;
            #Common_M_1_run.in_time.%X1 := TRUE;
            IF #Common_M_1_run.in_time.%X1 AND #Timer_M5000_run[1].Q THEN
                "P5204-DO" := TRUE;
                #Common_M_1_run.in_time.%X1 := FALSE;
                #Common_M_1_run.step := 16;
                RETURN;
            END_IF;
        END_IF;
        IF "P5204-DO" THEN
            #Common_M_1_run.step := 16;
        END_IF;
    END_IF;
    //step16
    IF #Common_M_1_run.step = 16 THEN
        IF NOT "P5104-DO" THEN
            IF #Common_M_1_run.todo THEN
                "P5104-DO" := TRUE;
                #Common_M_1_run.todo := FALSE;
                #Common_M_1_run.step := 17;
                RETURN;
            END_IF;
            #Common_M_1_run.in_time.%X1 := TRUE;
            IF #Common_M_1_run.in_time.%X1 AND #Timer_M5000_run[1].Q THEN
                "P5104-DO" := TRUE;
                #Common_M_1_run.in_time.%X1 := FALSE;
                #Common_M_1_run.step := 17;
                RETURN;
            END_IF;
        END_IF;
        IF "P5104-DO" THEN
            #Common_M_1_run.step := 17;
        END_IF;
    END_IF;
    //step17
    IF #Common_M_1_run.step = 17 THEN
        IF NOT "P5402-DO" THEN
            IF #Common_M_1_run.todo THEN
                "P5402-DO" := TRUE;
                #Common_M_1_run.todo := FALSE;
                #Common_M_1_run.step := 18;
                RETURN;
            END_IF;
            #Common_M_1_run.in_time.%X1 := TRUE;
            IF #Common_M_1_run.in_time.%X1 AND #Timer_M5000_run[1].Q THEN
                "P5402-DO" := TRUE;
                #Common_M_1_run.in_time.%X1 := FALSE;
                #Common_M_1_run.step := 18;
                RETURN;
            END_IF;
        END_IF;
        IF "P5402-DO" THEN
            #Common_M_1_run.step := 18;
        END_IF;
    END_IF;
    //step18
    IF #Common_M_1_run.step = 18 THEN
        IF NOT "P5302-DO" THEN
            IF #Common_M_1_run.todo THEN
                "P5302-DO" := TRUE;
                #Common_M_1_run.todo := FALSE;
                #Common_M_1_run.step := 19;
                RETURN;
            END_IF;
            #Common_M_1_run.in_time.%X1 := TRUE;
            IF #Common_M_1_run.in_time.%X1 AND #Timer_M5000_run[1].Q THEN
                "P5302-DO" := TRUE;
                #Common_M_1_run.in_time.%X1 := FALSE;
                #Common_M_1_run.step := 19;
                RETURN;
            END_IF;
        END_IF;
        IF "P5302-DO" THEN
            #Common_M_1_run.step := 19;
        END_IF;
    END_IF;
    //step19
    IF #Common_M_1_run.step = 19 THEN
        IF NOT "P5202-DO" THEN
            IF #Common_M_1_run.todo THEN
                "P5202-DO" := TRUE;
                #Common_M_1_run.todo := FALSE;
                #Common_M_1_run.step := 20;
                RETURN;
            END_IF;
            #Common_M_1_run.in_time.%X1 := TRUE;
            IF #Common_M_1_run.in_time.%X1 AND #Timer_M5000_run[1].Q THEN
                "P5202-DO" := TRUE;
                #Common_M_1_run.in_time.%X1 := FALSE;
                #Common_M_1_run.step := 20;
                RETURN;
            END_IF;
        END_IF;
        IF "P5202-DO" THEN
            #Common_M_1_run.step := 20;
        END_IF;
    END_IF;
    //step20
    IF #Common_M_1_run.step = 20 THEN
        IF NOT "P5102-DO" THEN
            IF #Common_M_1_run.todo THEN
                "P5102-DO" := TRUE;
                #Common_M_1_run.todo := FALSE;
                #Common_M_1_run.in_time := 0;
                #Common_M_1_run.step := 100;
                RETURN;
            END_IF;
            #Common_M_1_run.in_time.%X1 := TRUE;
            IF #Common_M_1_run.in_time.%X1 AND #Timer_M5000_run[1].Q THEN
                "P5102-DO" := TRUE;
                #Common_M_1_run.in_time := 0;
                #Common_M_1_run.step := 100;
                RETURN;
            END_IF;
        END_IF;
        IF "P5102-DO" THEN
            #Common_M_1_run.in_time := 0;
            #Common_M_1_run.step := 100;
        END_IF;
    END_IF;
    END_IF;
END_FUNCTION_BLOCK

(* ---- 11_15项目离心筛组控制程序修改.st ---- *)
REGION 预处理
    #"Motor-Runtimer"[0]( IN := #"Comm-run".busy, PT := #"Screen-Time"."PT-pretime-m");
    #"Motor-Runtimer"[1]( IN := #"Comm-run"."in-timer".%X1, PT := #"Screen-Time"."PT-runtime");
    #"Motor-Runtimer"[2]( IN := #"Comm-run"."in-timer".%X2, PT := #"Screen-Time"."PT-runtime");

    IF "Debug".Unit_estop_state[2] AND #bnt_manual THEN
        "Debug".Screen_state := 2;
        "Manual".M5101.man_enable := TRUE;
        "Manual".M5201.man_enable := TRUE;
        "Manual".M5002.man_enable := TRUE;
        "Manual".M5003.man_enable := TRUE;
        "Manual".M5004.man_enable := TRUE;
        "Manual".P5101.man_enable := TRUE;
        "Manual".P5102.man_enable := TRUE;
        "Manual".P5201.man_enable := TRUE;
        "Manual".P5202.man_enable := TRUE;
        "Manual".P5003.man_enable := TRUE;
        "Manual".P5004.man_enable := TRUE;
        "Manual".P5005.man_enable := TRUE;
        "Manual".P5006.man_enable := TRUE;
        "Manual".P5007.man_enable := TRUE;
        "Manual".P5008.man_enable := TRUE;
        "Manual".P5009.man_enable := TRUE;
        "Manual".P5010.man_enable := TRUE;
    END_IF;

    IF "Debug".Unit_estop_state[2] AND #bnt_auto THEN
        "Debug".Screen_state := 1;
        "Manual".M5101.man_enable := FALSE;
        "Manual".M5201.man_enable := FALSE;
        "Manual".M5002.man_enable := FALSE;
        "Manual".M5003.man_enable := FALSE;
        "Manual".M5004.man_enable := FALSE;
        "Manual".P5101.man_enable := FALSE;
        "Manual".P5102.man_enable := FALSE;
        "Manual".P5201.man_enable := FALSE;
        "Manual".P5202.man_enable := FALSE;
        "Manual".P5003.man_enable := FALSE;
        "Manual".P5004.man_enable := FALSE;
        "Manual".P5005.man_enable := FALSE;
        "Manual".P5006.man_enable := FALSE;
        "Manual".P5007.man_enable := FALSE;
        "Manual".P5008.man_enable := FALSE;
        "Manual".P5009.man_enable := FALSE;
        "Manual".P5010.man_enable := FALSE;
    END_IF;

    IF "Debug".Unit_estop_state[2] AND "Debug".Screen_state = 1 THEN
        IF #"Comm-run"."bnt-run" AND NOT #"Comm-run".busy THEN
            #"Comm-run".todo := 1;
            //复位工艺停止
            #"Comm-stop"."in-timer" := 0;
            #"Comm-stop".todo := 0;
            #"Comm-stop".busy := 0;
            #"Comm-stop".done := 0;
            #"Comm-stop".step := 0;
        END_IF;
        IF #"Comm-run".todo THEN
            #"Comm-run".busy := 1;
            #"Comm-run".step := 1;
            #"Comm-run".todo := 0;
        END_IF;
    ELSE
        #"Comm-run"."in-timer" := 0;
        #"Comm-run".todo := 0;
        #"Comm-run".busy := 0;
        #"Comm-run".done := 0;
        #"Comm-run".step := 0;
    END_IF;
END_REGION

REGION 工艺启动
    IF #"Comm-run".busy AND #"Motor-Runtimer"[0].Q THEN
        //step 1
        IF #"Comm-run".step = 1 THEN
            IF NOT "M5004-DO" THEN
                "M5004-DO" := 1;
                #"Comm-run"."in-timer".%X1 := 1;
                #"Comm-run".step := 2;
                RETURN;
            END_IF;
            IF "M5004-DO" THEN
                #"Comm-run".step := 2;
            END_IF;
        END_IF;
        //step 2
        IF #"Comm-run".step = 2 THEN
            IF NOT "M5003-DO" AND #"Comm-run"."in-timer".%X1 AND #"Motor-Runtimer"[1].Q THEN
                "M5003-DO" := 1;
                #"Comm-run"."in-timer".%X1 := 0;
                #"Comm-run"."in-timer".%X2 := 1;
                #"Comm-run".step := 3;
                RETURN;
            END_IF;
            IF NOT "M5003-DO" AND NOT #"Comm-run"."in-timer".%X1 THEN
                "M5003-DO" := 1;
                #"Comm-run"."in-timer".%X2 := 1;
                #"Comm-run".step := 3;
                RETURN;
            END_IF;
            IF "M5003-DO" THEN
                #"Comm-run".step := 3;
            END_IF;
        END_IF;
        //step 3
        IF #"Comm-run".step = 3 THEN
            IF NOT "M5002-DO" AND (#"Comm-run"."in-timer".%X1 )AND (#"Motor-Runtimer"[1].Q ) THEN
                "M5002-DO" := 1;
                #"Comm-run"."in-timer".%X1 := 0;
                #"Comm-run"."in-timer".%X2 := 1;
                #"Comm-run".step := 4;
                RETURN;
            END_IF;
            IF NOT "M5002-DO" AND (#"Comm-run"."in-timer".%X2)AND (#"Motor-Runtimer"[2].Q) THEN
                "M5002-DO" := 1;
                #"Comm-run"."in-timer".%X1 := 1;
                #"Comm-run"."in-timer".%X2 := 0;
                #"Comm-run".step := 4;
                RETURN;
            END_IF;
            IF NOT "M5002-DO" AND NOT (#"Comm-run"."in-timer".%X1 OR #"Comm-run"."in-timer".%X2) THEN
                "M5002-DO" := 1;
                #"Comm-run"."in-timer".%X1 := 1;
                #"Comm-run".step := 4;
                RETURN;
            END_IF;
            IF "M5002-DO" THEN
                #"Comm-run".step := 4;
            END_IF;
        END_IF;
        //step 4
        IF #"Comm-run".step = 4 THEN
            IF NOT "M5201-DO" AND (#"Comm-run"."in-timer".%X1 )AND (#"Motor-Runtimer"[1].Q ) THEN
                "M5201-DO" := 1;
                #"Comm-run"."in-timer".%X1 := 0;
                #"Comm-run"."in-timer".%X2 := 1;
                #"Comm-run".step := 5;
                RETURN;
            END_IF;
            IF NOT "M5201-DO" AND (#"Comm-run"."in-timer".%X2)AND (#"Motor-Runtimer"[2].Q) THEN
                "M5201-DO" := 1;
                #"Comm-run"."in-timer".%X1 := 1;
                #"Comm-run"."in-timer".%X2 := 0;
                #"Comm-run".step := 5;
                RETURN;
            END_IF;
            IF NOT "M5201-DO" AND NOT (#"Comm-run"."in-timer".%X1 OR #"Comm-run"."in-timer".%X2) THEN
                "M5201-DO" := 1;
                #"Comm-run"."in-timer".%X2 := 1;
                #"Comm-run".step := 5;
                RETURN;
            END_IF;
            IF "M5201-DO" THEN
                #"Comm-run".step := 5;
            END_IF;
        END_IF;
        //step 5
        IF #"Comm-run".step = 5 THEN
            IF NOT "M5101-DO" AND (#"Comm-run"."in-timer".%X1 )AND (#"Motor-Runtimer"[1].Q ) THEN
                "M5101-DO" := 1;
                #"Comm-run"."in-timer".%X1 := 0;
                #"Comm-run"."in-timer".%X2 := 1;
                #"Comm-run".step := 6;
                RETURN;
            END_IF;
            IF NOT "M5101-DO" AND (#"Comm-run"."in-timer".%X2)AND (#"Motor-Runtimer"[2].Q) THEN
                "M5101-DO" := 1;
                #"Comm-run"."in-timer".%X1 := 1;
                #"Comm-run"."in-timer".%X2 := 0;
                #"Comm-run".step := 6;
                RETURN;
            END_IF;
            IF NOT "M5101-DO" AND NOT (#"Comm-run"."in-timer".%X1 OR #"Comm-run"."in-timer".%X2) THEN
                "M5101-DO" := 1;
                #"Comm-run"."in-timer".%X1 := 1;
                #"Comm-run".step := 6;
                RETURN;
            END_IF;
            IF "M5101-DO" THEN
                #"Comm-run".step := 6;
            END_IF;
        END_IF;
        //step 6
        IF #"Comm-run".step = 6 THEN
            IF NOT "P5010-DO" AND (#"Comm-run"."in-timer".%X1 )AND (#"Motor-Runtimer"[1].Q ) THEN
                "P5010-DO" := 1;
                #"Comm-run"."in-timer".%X1 := 0;
                #"Comm-run"."in-timer".%X2 := 1;
                #"Comm-run".step := 7;
                RETURN;
            END_IF;
            IF NOT "P5010-DO" AND (#"Comm-run"."in-timer".%X2)AND (#"Motor-Runtimer"[2].Q) THEN
                "P5010-DO" := 1;
                #"Comm-run"."in-timer".%X1 := 1;
                #"Comm-run"."in-timer".%X2 := 0;
                #"Comm-run".step := 7;
                RETURN;
            END_IF;
            IF NOT "P5010-DO" AND NOT (#"Comm-run"."in-timer".%X1 OR #"Comm-run"."in-timer".%X2) THEN
                "P5010-DO" := 1;
                #"Comm-run"."in-timer".%X2 := 1;
                #"Comm-run".step := 7;
                RETURN;
            END_IF;
            IF "P5010-DO" THEN
                #"Comm-run".step := 7;
            END_IF;
        END_IF;
        //step 7
        IF #"Comm-run".step = 7 THEN
            IF NOT "P5007-DO" AND (#"Comm-run"."in-timer".%X1 )AND (#"Motor-Runtimer"[1].Q ) THEN
                "P5007-DO" := 1;
                #"Comm-run"."in-timer".%X1 := 0;
                #"Comm-run"."in-timer".%X2 := 1;
                #"Comm-run".step := 8;
                RETURN;
            END_IF;
            IF NOT "P5007-DO" AND (#"Comm-run"."in-timer".%X2)AND (#"Motor-Runtimer"[2].Q) THEN
                "P5007-DO" := 1;
                #"Comm-run"."in-timer".%X1 := 1;
                #"Comm-run"."in-timer".%X2 := 0;
                #"Comm-run".step := 8;
                RETURN;
            END_IF;
            IF NOT "P5007-DO" AND NOT (#"Comm-run"."in-timer".%X1 OR #"Comm-run"."in-timer".%X2) THEN
                "P5007-DO" := 1;
                #"Comm-run"."in-timer".%X1 := 1;
                #"Comm-run".step := 8;
                RETURN;
            END_IF;
            IF "P5007-DO" THEN
                #"Comm-run".step := 8;
            END_IF;
        END_IF;
        //step 8
        IF #"Comm-run".step = 8 THEN
            IF NOT "P5005-DO" AND (#"Comm-run"."in-timer".%X1 )AND (#"Motor-Runtimer"[1].Q ) THEN
                "P5005-DO" := 1;
                #"Comm-run"."in-timer".%X1 := 0;
                #"Comm-run"."in-timer".%X2 := 1;
                #"Comm-run".step := 9;
                RETURN;
            END_IF;
            IF NOT "P5005-DO" AND (#"Comm-run"."in-timer".%X2)AND (#"Motor-Runtimer"[2].Q) THEN
                "P5005-DO" := 1;
                #"Comm-run"."in-timer".%X1 := 1;
                #"Comm-run"."in-timer".%X2 := 0;
                #"Comm-run".step := 9;
                RETURN;
            END_IF;
            IF NOT "P5005-DO" AND NOT (#"Comm-run"."in-timer".%X1 OR #"Comm-run"."in-timer".%X2) THEN
                "P5005-DO" := 1;
                #"Comm-run"."in-timer".%X2 := 1;
                #"Comm-run".step := 9;
                RETURN;
            END_IF;
            IF "P5005-DO" THEN
                #"Comm-run".step := 9;
            END_IF;
        END_IF;
        //step 9
        IF #"Comm-run".step = 9 THEN
            IF NOT "P5003-DO" AND (#"Comm-run"."in-timer".%X1 )AND (#"Motor-Runtimer"[1].Q ) THEN
                "P5003-DO" := 1;
                #"Comm-run"."in-timer".%X1 := 0;
                #"Comm-run"."in-timer".%X2 := 1;
                #"Comm-run".step := 10;
                RETURN;
            END_IF;
            IF NOT "P5003-DO" AND (#"Comm-run"."in-timer".%X2)AND (#"Motor-Runtimer"[2].Q) THEN
                "P5003-DO" := 1;
                #"Comm-run"."in-timer".%X1 := 1;
                #"Comm-run"."in-timer".%X2 := 0;
                #"Comm-run".step := 10;
                RETURN;
            END_IF;
            IF NOT "P5003-DO" AND NOT (#"Comm-run"."in-timer".%X1 OR #"Comm-run"."in-timer".%X2) THEN
                "P5003-DO" := 1;
                #"Comm-run"."in-timer".%X1 := 1;
                #"Comm-run".step := 10;
                RETURN;
            END_IF;
            IF "P5003-DO" THEN
                #"Comm-run".step := 10;
            END_IF;
        END_IF;
        //step 10
        IF #"Comm-run".step = 10 THEN
            IF NOT "P5201-DO" AND (#"Comm-run"."in-timer".%X1 )AND (#"Motor-Runtimer"[1].Q ) THEN
                "P5201-DO" := 1;
                #"Comm-run"."in-timer".%X1 := 0;
                #"Comm-run"."in-timer".%X2 := 1;
                #"Comm-run".step := 11;
                RETURN;
            END_IF;
            IF NOT "P5201-DO" AND (#"Comm-run"."in-timer".%X2) AND (#"Motor-Runtimer"[2].Q) THEN
                "P5201-DO" := 1;
                #"Comm-run"."in-timer".%X1 := 1;
                #"Comm-run"."in-timer".%X2 := 0;
                #"Comm-run".step := 11;
                RETURN;
            END_IF;
            IF NOT "P5201-DO" AND NOT (#"Comm-run"."in-timer".%X1 OR #"Comm-run"."in-timer".%X2) THEN
                "P5201-DO" := 1;
                #"Comm-run"."in-timer".%X2 := 1;
                #"Comm-run".step := 11;
                RETURN;
            END_IF;
            IF "P5201-DO" THEN
                #"Comm-run".step := 11;
            END_IF;
        END_IF;
        //step 11
        IF #"Comm-run".step = 11 THEN
            IF NOT "P5101-DO" AND (#"Comm-run"."in-timer".%X1 )AND (#"Motor-Runtimer"[1].Q ) THEN
                "P5101-DO" := 1;
                #"Comm-run"."in-timer".%X1 := 0;
                #"Comm-run"."in-timer".%X2 := 1;
                #"Comm-run".step := 12;
                RETURN;
            END_IF;
            IF NOT "P5101-DO" AND (#"Comm-run"."in-timer".%X2) AND (#"Motor-Runtimer"[2].Q) THEN
                "P5101-DO" := 1;
                #"Comm-run"."in-timer".%X1 := 1;
                #"Comm-run"."in-timer".%X2 := 0;
                #"Comm-run".step := 12;
                RETURN;
            END_IF;
            IF NOT "P5101-DO" AND NOT (#"Comm-run"."in-timer".%X1 OR #"Comm-run"."in-timer".%X2) THEN
                "P5101-DO" := 1;
                #"Comm-run"."in-timer".%X1 := 1;
                #"Comm-run".step := 12;
                RETURN;
            END_IF;
            IF "P5101-DO" THEN
                #"Comm-run".step := 12;
            END_IF;
        END_IF;
        //step 12
        IF #"Comm-run".step = 12 THEN
            IF NOT "P5009-DO" AND (#"Comm-run"."in-timer".%X1 )AND (#"Motor-Runtimer"[1].Q ) THEN
                "P5009-DO" := 1;
                #"Comm-run"."in-timer".%X1 := 0;
                #"Comm-run"."in-timer".%X2 := 1;
                #"Comm-run".step := 13;
                RETURN;
            END_IF;
            IF NOT "P5009-DO" AND (#"Comm-run"."in-timer".%X2) AND (#"Motor-Runtimer"[2].Q) THEN
                "P5009-DO" := 1;
                #"Comm-run"."in-timer".%X1 := 1;
                #"Comm-run"."in-timer".%X2 := 0;
                #"Comm-run".step := 13;
                RETURN;
            END_IF;
            IF NOT "P5009-DO" AND NOT (#"Comm-run"."in-timer".%X1 OR #"Comm-run"."in-timer".%X2) THEN
                "P5009-DO" := 1;
                #"Comm-run"."in-timer".%X2 := 1;
                #"Comm-run".step := 13;
                RETURN;
            END_IF;
            IF "P5009-DO" THEN
                #"Comm-run".step := 13;
            END_IF;
        END_IF;
        //step 13
        IF #"Comm-run".step = 13 THEN
            IF NOT "P5008-DO" AND (#"Comm-run"."in-timer".%X1 )AND (#"Motor-Runtimer"[1].Q ) THEN
                "P5008-DO" := 1;
                #"Comm-run"."in-timer".%X1 := 0;
                #"Comm-run"."in-timer".%X2 := 1;
                #"Comm-run".step := 14;
                RETURN;
            END_IF;
            IF NOT "P5008-DO" AND (#"Comm-run"."in-timer".%X2) AND (#"Motor-Runtimer"[2].Q) THEN
                "P5008-DO" := 1;
                #"Comm-run"."in-timer".%X1 := 1;
                #"Comm-run"."in-timer".%X2 := 0;
                #"Comm-run".step := 14;
                RETURN;
            END_IF;
            IF NOT "P5008-DO" AND NOT (#"Comm-run"."in-timer".%X1 OR #"Comm-run"."in-timer".%X2) THEN
                "P5008-DO" := 1;
                #"Comm-run"."in-timer".%X1 := 1;
                #"Comm-run".step := 14;
                RETURN;
            END_IF;
            IF "P5008-DO" THEN
                #"Comm-run".step := 14;
            END_IF;
        END_IF;
        //step 14
        IF #"Comm-run".step = 14 THEN
            IF NOT "P5006-DO" AND (#"Comm-run"."in-timer".%X1 )AND (#"Motor-Runtimer"[1].Q ) THEN
                "P5006-DO" := 1;
                #"Comm-run"."in-timer".%X1 := 0;
                #"Comm-run"."in-timer".%X2 := 1;
                #"Comm-run".step := 15;
                RETURN;
            END_IF;
            IF NOT "P5006-DO" AND (#"Comm-run"."in-timer".%X2) AND (#"Motor-Runtimer"[2].Q) THEN
                "P5006-DO" := 1;
                #"Comm-run"."in-timer".%X1 := 1;
                #"Comm-run"."in-timer".%X2 := 0;
                #"Comm-run".step := 15;
                RETURN;
            END_IF;
            IF NOT "P5006-DO" AND NOT (#"Comm-run"."in-timer".%X1 OR #"Comm-run"."in-timer".%X2) THEN
                "P5006-DO" := 1;
                #"Comm-run"."in-timer".%X2 := 1;
                #"Comm-run".step := 15;
                RETURN;
            END_IF;
            IF "P5006-DO" THEN
                #"Comm-run".step := 15;
            END_IF;
        END_IF;
        //step 15
        IF #"Comm-run".step = 15 THEN
            IF NOT "P5004-DO" AND (#"Comm-run"."in-timer".%X1 )AND (#"Motor-Runtimer"[1].Q ) THEN
                "P5004-DO" := 1;
                #"Comm-run"."in-timer".%X1 := 0;
                #"Comm-run"."in-timer".%X2 := 1;
                #"Comm-run".step := 16;
                RETURN;
            END_IF;
            IF NOT "P5004-DO" AND (#"Comm-run"."in-timer".%X2) AND (#"Motor-Runtimer"[2].Q) THEN
                "P5004-DO" := 1;
                #"Comm-run"."in-timer".%X1 := 1;
                #"Comm-run"."in-timer".%X2 := 0;
                #"Comm-run".step := 16;
                RETURN;
            END_IF;
            IF NOT "P5004-DO" AND NOT (#"Comm-run"."in-timer".%X1 OR #"Comm-run"."in-timer".%X2) THEN
                "P5004-DO" := 1;
                #"Comm-run"."in-timer".%X2 := 1;
                #"Comm-run".step := 16;
                RETURN;
            END_IF;
            IF "P5004-DO" THEN
                #"Comm-run".step := 16;
            END_IF;
        END_IF;
        //step 16
        IF #"Comm-run".step = 16 THEN
            IF NOT "P5202-DO" AND (#"Comm-run"."in-timer".%X1 )AND (#"Motor-Runtimer"[1].Q ) THEN
                "P5202-DO" := 1;
                #"Comm-run"."in-timer".%X1 := 0;
                #"Comm-run"."in-timer".%X2 := 1;
                #"Comm-run".step := 17;
                RETURN;
            END_IF;
            IF NOT "P5202-DO" AND (#"Comm-run"."in-timer".%X2) AND (#"Motor-Runtimer"[2].Q) THEN
                "P5202-DO" := 1;
                #"Comm-run"."in-timer".%X1 := 1;
                #"Comm-run"."in-timer".%X2 := 0;
                #"Comm-run".step := 17;
                RETURN;
            END_IF;
            IF NOT "P5202-DO" AND NOT (#"Comm-run"."in-timer".%X1 OR #"Comm-run"."in-timer".%X2) THEN
                "P5202-DO" := 1;
                #"Comm-run"."in-timer".%X2 := 1;
                #"Comm-run".step := 17;
                RETURN;
            END_IF;
            IF "P5202-DO" THEN
                #"Comm-run".step := 17;
            END_IF;
        END_IF;
        //step 17
        IF #"Comm-run".step = 17 THEN
            IF NOT "P5102-DO" AND (#"Comm-run"."in-timer".%X1 )AND (#"Motor-Runtimer"[1].Q ) THEN
                "P5102-DO" := 1;
                #"Comm-run"."in-timer".%X1 := 0;
                #"Comm-run".step := 18;
                RETURN;
            END_IF;
            IF NOT "P5102-DO" AND (#"Comm-run"."in-timer".%X2) AND (#"Motor-Runtimer"[2].Q) THEN
                "P5102-DO" := 1;
                #"Comm-run"."in-timer".%X2 := 0;
                #"Comm-run".step := 18;
                RETURN;
            END_IF;
            IF NOT "P5102-DO" AND NOT (#"Comm-run"."in-timer".%X1 OR #"Comm-run"."in-timer".%X2) THEN
                "P5102-DO" := 1;
                #"Comm-run".step := 18;
                RETURN;
            END_IF;
            IF "P5102-DO" THEN
                #"Comm-run".step := 18;
            END_IF;
        END_IF;
        //step 18
        IF #"Comm-run".step = 18 THEN
            #"Comm-run"."in-timer" := 0;
            #"Comm-run".todo := 0;
            #"Comm-run".busy := 0;
            #"Comm-run".done := 1;
        END_IF;

    END_IF;

REGION 工艺停止
    IF #"Comm-stop".busy AND #"Motor-Stoptimer"[0].Q THEN
        //step 1
        IF #"Comm-stop".step = 1 THEN
            IF "P5102-DO" THEN
                "P5102-DO" := 0;
                #"Comm-stop"."in-timer".%X1 := 1;
                #"Comm-stop".step := 2;
                RETURN;
            END_IF;
            IF NOT "P5102-DO" THEN
                #"Comm-stop".step := 2;
            END_IF;
        END_IF;
        //step 2
        IF #"Comm-stop".step = 2 THEN
            IF "P5202-DO" AND #"Comm-stop"."in-timer".%X1 AND #"Motor-Stoptimer"[1].Q THEN
                "P5202-DO" := 0;
                #"Comm-stop"."in-timer".%X1 := 0;
                #"Comm-stop"."in-timer".%X2 := 1;
                #"Comm-stop".step := 3;
                RETURN;
            END_IF;
            IF "P5202-DO" AND NOT #"Comm-stop"."in-timer".%X1 THEN
                "P5202-DO" := 0;
                #"Comm-stop"."in-timer".%X2 := 1;
                #"Comm-stop".step := 3;
                RETURN;
            END_IF;
            IF NOT "P5202-DO" THEN
                #"Comm-stop".step := 3;
            END_IF;
        END_IF;
        //step 3
        IF #"Comm-stop".step = 3 THEN
            IF "P5004-DO" AND (#"Comm-stop"."in-timer".%X1 OR #"Comm-stop"."in-timer".%X2)
                AND (#"Motor-Stoptimer"[1].Q OR #"Motor-Stoptimer"[2].Q) THEN
                "P5004-DO" := 0;
                #"Comm-stop"."in-timer".%X1 := 1;
                #"Comm-stop"."in-timer".%X2 := 0;
                #"Comm-stop".step := 4;
                RETURN;
            END_IF;
            IF "P5004-DO" AND NOT (#"Comm-stop"."in-timer".%X1 OR #"Comm-stop"."in-timer".%X2) THEN
                "P5004-DO" := 0;
                #"Comm-stop"."in-timer".%X1 := 1;
                #"Comm-stop".step := 4;
                RETURN;
            END_IF;
            IF NOT "P5004-DO" THEN
                #"Comm-stop".step := 4;
            END_IF;
        END_IF;
        //step 4
        IF #"Comm-stop".step = 4 THEN
            IF "P5006-DO" AND (#"Comm-stop"."in-timer".%X1 OR #"Comm-stop"."in-timer".%X2)
                AND (#"Motor-Stoptimer"[1].Q OR #"Motor-Stoptimer"[2].Q) THEN
                "P5006-DO" := 0;
                #"Comm-stop"."in-timer".%X1 := 0;
                #"Comm-stop"."in-timer".%X2 := 1;
                #"Comm-stop".step := 5;
                RETURN;
            END_IF;
            IF "P5006-DO" AND NOT (#"Comm-stop"."in-timer".%X1 OR #"Comm-stop"."in-timer".%X2) THEN
                "P5006-DO" := 0;
                #"Comm-stop"."in-timer".%X2 := 1;
                #"Comm-stop".step := 5;
                RETURN;
            END_IF;
            IF NOT "P5006-DO" THEN
                #"Comm-stop".step := 5;
            END_IF;
        END_IF;
        //step 5
        IF #"Comm-stop".step = 5 THEN
            IF "P5008-DO" AND (#"Comm-stop"."in-timer".%X1 OR #"Comm-stop"."in-timer".%X2)
                AND (#"Motor-Stoptimer"[1].Q OR #"Motor-Stoptimer"[2].Q) THEN
                "P5008-DO" := 0;
                #"Comm-stop"."in-timer".%X1 := 1;
                #"Comm-stop"."in-timer".%X2 := 0;
                #"Comm-stop".step := 6;
                RETURN;
            END_IF;
            IF "P5008-DO" AND NOT (#"Comm-stop"."in-timer".%X1 OR #"Comm-stop"."in-timer".%X2) THEN
                "P5008-DO" := 0;
                #"Comm-stop"."in-timer".%X1 := 1;
                #"Comm-stop".step := 6;
                RETURN;
            END_IF;
            IF NOT "P5008-DO" THEN
                #"Comm-stop".step := 6;
            END_IF;
        END_IF;
        //step 6
        IF #"Comm-stop".step = 6 THEN
            IF "P5009-DO" AND (#"Comm-stop"."in-timer".%X1 OR #"Comm-stop"."in-timer".%X2)
                AND (#"Motor-Stoptimer"[1].Q OR #"Motor-Stoptimer"[2].Q) THEN
                "P5009-DO" := 0;
                #"Comm-stop"."in-timer".%X1 := 0;
                #"Comm-stop"."in-timer".%X2 := 1;
                #"Comm-stop".step := 7;
                RETURN;
            END_IF;
            IF "P5009-DO" AND NOT (#"Comm-stop"."in-timer".%X1 OR #"Comm-stop"."in-timer".%X2) THEN
                "P5009-DO" := 0;
                #"Comm-stop"."in-timer".%X2 := 1;
                #"Comm-stop".step := 7;
                RETURN;
            END_IF;
            IF NOT "P5009-DO" THEN
                #"Comm-stop".step := 7;
            END_IF;
        END_IF;
        //step 7
        IF #"Comm-stop".step = 7 THEN
            IF "P5101-DO" AND (#"Comm-stop"."in-timer".%X1 OR #"Comm-stop"."in-timer".%X2)
                AND (#"Motor-Stoptimer"[1].Q OR #"Motor-Stoptimer"[2].Q) THEN
                "P5101-DO" := 0;
                #"Comm-stop"."in-timer".%X1 := 1;
                #"Comm-stop"."in-timer".%X2 := 0;
                #"Comm-stop".step := 8;
                RETURN;
            END_IF;
            IF "P5101-DO" AND NOT (#"Comm-stop"."in-timer".%X1 OR #"Comm-stop"."in-timer".%X2) THEN
                "P5101-DO" := 0;
                #"Comm-stop"."in-timer".%X1 := 1;
                #"Comm-stop".step := 8;
                RETURN;
            END_IF;
            IF NOT "P5101-DO" THEN
                #"Comm-stop".step := 8;
            END_IF;
        END_IF;
        //step 8
        IF #"Comm-stop".step = 8 THEN
            IF "P5201-DO" AND (#"Comm-stop"."in-timer".%X1 OR #"Comm-stop"."in-timer".%X2)
                AND (#"Motor-Stoptimer"[1].Q OR #"Motor-Stoptimer"[2].Q) THEN
                "P5201-DO" := 0;
                #"Comm-stop"."in-timer".%X1 := 0;
                #"Comm-stop"."in-timer".%X2 := 1;
                #"Comm-stop".step := 9;
                RETURN;
            END_IF;
            IF "P5201-DO" AND NOT (#"Comm-stop"."in-timer".%X1 OR #"Comm-stop"."in-timer".%X2) THEN
                "P5201-DO" := 0;
                #"Comm-stop"."in-timer".%X2 := 1;
                #"Comm-stop".step := 9;
                RETURN;
            END_IF;
            IF NOT "P5201-DO" THEN
                #"Comm-stop".step := 9;
            END_IF;
        END_IF;
        //step 9
        IF #"Comm-stop".step = 9 THEN
            IF "P5003-DO" AND (#"Comm-stop"."in-timer".%X1 OR #"Comm-stop"."in-timer".%X2)
                AND (#"Motor-Stoptimer"[1].Q OR #"Motor-Stoptimer"[2].Q) THEN
                "P5003-DO" := 0;
                #"Comm-stop"."in-timer".%X1 := 1;
                #"Comm-stop"."in-timer".%X2 := 0;
                #"Comm-stop".step := 10;
                RETURN;
            END_IF;
            IF "P5003-DO" AND NOT (#"Comm-stop"."in-timer".%X1 OR #"Comm-stop"."in-timer".%X2) THEN
                "P5003-DO" := 0;
                #"Comm-stop"."in-timer".%X1 := 1;
                #"Comm-stop".step := 10;
                RETURN;
            END_IF;
            IF NOT "P5003-DO" THEN
                #"Comm-stop".step := 10;
            END_IF;
        END_IF;
        //step 10
        IF #"Comm-stop".step = 10 THEN
            IF "P5005-DO" AND (#"Comm-stop"."in-timer".%X1 OR #"Comm-stop"."in-timer".%X2)
                AND (#"Motor-Stoptimer"[1].Q OR #"Motor-Stoptimer"[2].Q) THEN
                "P5005-DO" := 0;
                #"Comm-stop"."in-timer".%X1 := 0;
                #"Comm-stop"."in-timer".%X2 := 1;
                #"Comm-stop".step := 11;
                RETURN;
            END_IF;
            IF "P5005-DO" AND NOT (#"Comm-stop"."in-timer".%X1 OR #"Comm-stop"."in-timer".%X2) THEN
                "P5005-DO" := 0;
                #"Comm-stop"."in-timer".%X2 := 1;
                #"Comm-stop".step := 11;
                RETURN;
            END_IF;
            IF NOT "P5005-DO" THEN
                #"Comm-stop".step := 11;
            END_IF;
        END_IF;
        //step 11
        IF #"Comm-stop".step = 11 THEN
            IF "P5007-DO" AND (#"Comm-stop"."in-timer".%X1 OR #"Comm-stop"."in-timer".%X2)
                AND (#"Motor-Stoptimer"[1].Q OR #"Motor-Stoptimer"[2].Q) THEN
                "P5007-DO" := 0;
                #"Comm-stop"."in-timer".%X1 := 1;
                #"Comm-stop"."in-timer".%X2 := 0;
                #"Comm-stop".step := 12;
                RETURN;
            END_IF;
            IF "P5007-DO" AND NOT (#"Comm-stop"."in-timer".%X1 OR #"Comm-stop"."in-timer".%X2) THEN
                "P5007-DO" := 0;
                #"Comm-stop"."in-timer".%X1 := 1;
                #"Comm-stop".step := 12;
                RETURN;
            END_IF;
            IF NOT "P5007-DO" THEN
                #"Comm-stop".step := 12;
            END_IF;
        END_IF;
        //step 12
        IF #"Comm-stop".step = 12 THEN
            IF "P5010-DO" AND (#"Comm-stop"."in-timer".%X1 OR #"Comm-stop"."in-timer".%X2)
                AND (#"Motor-Stoptimer"[1].Q OR #"Motor-Stoptimer"[2].Q) THEN
                "P5010-DO" := 0;
                #"Comm-stop"."in-timer".%X1 := 0;
                #"Comm-stop"."in-timer".%X2 := 1;
                #"Comm-stop".step := 13;
                RETURN;
            END_IF;
            IF "P5010-DO" AND NOT (#"Comm-stop"."in-timer".%X1 OR #"Comm-stop"."in-timer".%X2) THEN
                "P5010-DO" := 0;
                #"Comm-stop"."in-timer".%X2 := 1;
                #"Comm-stop".step := 13;
                RETURN;
            END_IF;
            IF NOT "P5010-DO" THEN
                #"Comm-stop".step := 13;
            END_IF;
        END_IF;
        //step 13
        IF #"Comm-stop".step = 13 THEN
            IF "M5101-DO" AND (#"Comm-stop"."in-timer".%X1 OR #"Comm-stop"."in-timer".%X2)
                AND (#"Motor-Stoptimer"[1].Q OR #"Motor-Stoptimer"[2].Q) THEN
                "M5101-DO" := 0;
                #"Comm-stop"."in-timer".%X1 := 1;
                #"Comm-stop"."in-timer".%X2 := 0;
                #"Comm-stop".step := 14;
                RETURN;
            END_IF;
            IF "M5101-DO" AND NOT (#"Comm-stop"."in-timer".%X1 OR #"Comm-stop"."in-timer".%X2) THEN
                "M5101-DO" := 0;
                #"Comm-stop"."in-timer".%X1 := 1;
                #"Comm-stop".step := 14;
                RETURN;
            END_IF;
            IF NOT "M5101-DO" THEN
                #"Comm-stop".step := 14;
            END_IF;
        END_IF;
        //step 14
        IF #"Comm-stop".step = 14 THEN
            IF "M5201-DO" AND (#"Comm-stop"."in-timer".%X1 OR #"Comm-stop"."in-timer".%X2)
                AND (#"Motor-Stoptimer"[1].Q OR #"Motor-Stoptimer"[2].Q) THEN
                "M5201-DO" := 0;
                #"Comm-stop"."in-timer".%X1 := 0;
                #"Comm-stop"."in-timer".%X2 := 1;
                #"Comm-stop".step := 15;
                RETURN;
            END_IF;
            IF "M5201-DO" AND NOT (#"Comm-stop"."in-timer".%X1 OR #"Comm-stop"."in-timer".%X2) THEN
                "M5201-DO" := 0;
                #"Comm-stop"."in-timer".%X2 := 1;
                #"Comm-stop".step := 15;
                RETURN;
            END_IF;
            IF NOT "M5201-DO" THEN
                #"Comm-stop".step := 15;
            END_IF;
        END_IF;
        //step 15
        IF #"Comm-stop".step = 15 THEN
            IF "M5002-DO" AND (#"Comm-stop"."in-timer".%X1 OR #"Comm-stop"."in-timer".%X2)
                AND (#"Motor-Stoptimer"[1].Q OR #"Motor-Stoptimer"[2].Q) THEN
                "M5002-DO" := 0;
                #"Comm-stop"."in-timer".%X1 := 1;
                #"Comm-stop"."in-timer".%X2 := 0;
                #"Comm-stop".step := 16;
                RETURN;
            END_IF;
            IF "M5002-DO" AND NOT (#"Comm-stop"."in-timer".%X1 OR #"Comm-stop"."in-timer".%X2) THEN
                "M5002-DO" := 0;
                #"Comm-stop"."in-timer".%X1 := 1;
                #"Comm-stop".step := 16;
                RETURN;
            END_IF;
            IF NOT "M5002-DO" THEN
                #"Comm-stop".step := 16;
            END_IF;
        END_IF;
        //step 16
        IF #"Comm-stop".step = 16 THEN
            IF "M5003-DO" AND (#"Comm-stop"."in-timer".%X1 OR #"Comm-stop"."in-timer".%X2)
                AND (#"Motor-Stoptimer"[1].Q OR #"Motor-Stoptimer"[2].Q) THEN
                "M5003-DO" := 0;
                #"Comm-stop"."in-timer".%X1 := 0;
                #"Comm-stop"."in-timer".%X2 := 1;
                #"Comm-stop".step := 17;
                RETURN;
            END_IF;
            IF "M5003-DO" AND NOT (#"Comm-stop"."in-timer".%X1 OR #"Comm-stop"."in-timer".%X2) THEN
                "M5003-DO" := 0;
                #"Comm-stop"."in-timer".%X2 := 1;
                #"Comm-stop".step := 17;
                RETURN;
            END_IF;
            IF NOT "M5003-DO" THEN
                #"Comm-stop".step := 17;
            END_IF;
        END_IF;
        //step 17
        IF #"Comm-stop".step = 17 THEN
            IF "M5004-DO" AND (#"Comm-stop"."in-timer".%X1 OR #"Comm-stop"."in-timer".%X2)
                AND (#"Motor-Stoptimer"[1].Q OR #"Motor-Stoptimer"[2].Q) THEN
                "M5004-DO" := 0;
                #"Comm-stop".step := 18;
                RETURN;
            END_IF;
            IF "M5004-DO" AND NOT (#"Comm-stop"."in-timer".%X1 OR #"Comm-stop"."in-timer".%X2) THEN
                "M5004-DO" := 0;
                #"Comm-stop".step := 18;
                RETURN;
            END_IF;
            IF NOT "M5004-DO" THEN
                #"Comm-stop".step := 18;
            END_IF;
        END_IF;
        //step 18
        IF #"Comm-stop".step = 18 THEN
            #"Comm-stop"."in-timer" := 0;
            #"Comm-stop".todo := 0;
            #"Comm-stop".busy := 0;
            #"Comm-stop".done := 1;
        END_IF;

    END_IF;
END_REGION

(* ---- AI.st ---- *)
PROGRAM MainProgram;
VAR
    Motor1: BOOL; // 电机1的输出变量
    Motor2: BOOL; // 电机2的输出变量
    Motor3: BOOL; // 电机3的输出变量
END_VAR

// 电机启动顺序程序块
PROGRAM MotorStartupSequence;
VAR
    seqStep: INT; // 顺序步骤变量
END_VAR

// 顺序功能块，用于控制电机启动顺序
SEQ seqMotorStartup;

// 程序块主体
BEGIN
    seqMotorStartup(
        IN:= NOT seqMotorStartup.Q, // 当顺序功能块完成时，输入信号变为0
        Q0:= seqStep = 0, // 当顺序步骤为0时，输出Q0为1
        Q1:= seqStep = 1, // 当顺序步骤为1时，输出Q1为1
        Q2:= seqStep = 2  // 当顺序步骤为2时，输出Q2为1
    );

    // 根据顺序功能块的输出，控制电机的启动
    Motor1 := seqMotorStartup.Q0;
    Motor2 := seqMotorStartup.Q1;
    Motor3 := seqMotorStartup.Q2;

    // 如果所有电机都启动，增加顺序步骤
    IF seqMotorStartup.Q2 THEN
        seqStep := seqStep + 1;
    END_IF;
END_PROGRAM

// 主程序调用电机启动顺序程序块
BEGIN
    MotorStartupSequence();
END_PROGRAM

(* ---- ProcessRun.st ---- *)
REGION 预处理
    #"FP-run-bnt"(CLK:=#"Comm-run"."bnt-run");
    #"Motor-Runtimer"[0](IN := #"Comm-run".busy,
                         PT := #"Screen-Time"."PT-pretime-m");
    #"Motor-Runtimer"[1](IN := #"Comm-run"."in-timer".%X1,
                         PT := #"Screen-Time"."PT-runtime");
    #"Motor-Runtimer"[2](IN := #"Comm-run"."in-timer".%X2,
                         PT := #"Screen-Time"."PT-runtime");
    IF "Debug".Unit_estop_state[2] AND "Debug".Screen_state = 1 THEN
        IF #"FP-run-bnt".Q AND NOT #"Comm-run".busy THEN
            #"Comm-run".todo := 1;
            //复位工艺停止
            #"Comm-stop"."in-timer" := 0;
            #"Comm-stop".todo := 0;
            #"Comm-stop".busy := 0;
            #"Comm-stop".done := 0;
            #"Comm-stop".step := 0;
        END_IF;
        IF #"Comm-run".todo THEN
            #"Comm-run".busy := 1;
            #"Comm-run".step := 1;
            #"Comm-run".todo := 0;
        END_IF;
    ELSE
        #"Comm-run"."in-timer" := 0;
        #"Comm-run".todo := 0;
        #"Comm-run".busy := 0;
        #"Comm-run".done := 0;
        #"Comm-run".step := 0;
    END_IF;

END_REGION
REGION 工艺启动
    IF #"Comm-run".busy AND #"Motor-Runtimer"[0].Q THEN
        //step 1
        IF #"Comm-run".step = 1 THEN
            IF NOT "P5010-DO" THEN
                "P5010-DO" := 1;
                #"Comm-run"."in-timer".%X1 := 1;
                #"Comm-run".step := 2;
                RETURN;
            END_IF;
            IF "P5010-DO" THEN
                #"Comm-run".step := 2;
            END_IF;
        END_IF;
        //step 2
        IF #"Comm-run".step = 2 THEN
            IF NOT "P5009-DO" AND #"Comm-run"."in-timer".%X1 AND #"Motor-Runtimer"[1].Q THEN
                "P5009-DO" := 1;
                #"Comm-run"."in-timer".%X1 := 0;
                #"Comm-run"."in-timer".%X2 := 1;
                #"Comm-run".step := 3;
                RETURN;
            END_IF;
            IF NOT "P5009-DO" AND NOT #"Comm-run"."in-timer".%X1 THEN
                "P5009-DO" := 1;
                #"Comm-run"."in-timer".%X2 := 1;
                #"Comm-run".step := 3;
                RETURN;
            END_IF;
            IF "P5009-DO" THEN
                #"Comm-run".step := 3;
            END_IF;
        END_IF;
        //step 3
        IF #"Comm-run".step = 3 THEN
            IF NOT "M5201-DO" AND (#"Comm-run"."in-timer".%X1 OR #"Comm-run"."in-timer".%X2)
                AND (#"Motor-Runtimer"[1].Q OR #"Motor-Runtimer"[2].Q) THEN
                "M5201-DO" := 1;
                #"Comm-run"."in-timer".%X1 := 1;
                #"Comm-run"."in-timer".%X2 := 0;
                #"Comm-run".step := 4;
                RETURN;
            END_IF;
            IF NOT "M5201-DO" AND NOT (#"Comm-run"."in-timer".%X1 OR #"Comm-run"."in-timer".%X2) THEN
                "M5201-DO" := 1;
                #"Comm-run"."in-timer".%X1 := 1;
                #"Comm-run".step := 4;
                RETURN;
            END_IF;
            IF "M5201-DO" THEN
                #"Comm-run".step := 4;
            END_IF;
        END_IF;
        //step 4
        IF #"Comm-run".step = 4 THEN
            IF NOT "P5002-DO" AND (#"Comm-run"."in-timer".%X1 OR #"Comm-run"."in-timer".%X2)
                AND (#"Motor-Runtimer"[1].Q OR #"Motor-Runtimer"[2].Q) THEN
                "P5002-DO" := 1;
                #"Comm-run"."in-timer".%X1 := 0;
                #"Comm-run"."in-timer".%X2 := 1;
                #"Comm-run".step := 5;
                RETURN;
            END_IF;
            IF NOT "P5002-DO" AND NOT (#"Comm-run"."in-timer".%X1 OR #"Comm-run"."in-timer".%X2) THEN
                "P5002-DO" := 1;
                #"Comm-run"."in-timer".%X2 := 1;
                #"Comm-run".step := 5;
                RETURN;
            END_IF;
            IF "P5002-DO" THEN
                #"Comm-run".step := 5;
            END_IF;
        END_IF;
        //step 5
        IF #"Comm-run".step = 5 THEN
            IF NOT "P5001-DO" AND (#"Comm-run"."in-timer".%X1 OR #"Comm-run"."in-timer".%X2)
                AND (#"Motor-Runtimer"[1].Q OR #"Motor-Runtimer"[2].Q) THEN
                "P5001-DO" := 1;
                #"Comm-run"."in-timer".%X1 := 1;
                #"Comm-run"."in-timer".%X2 := 0;
                #"Comm-run".step := 6;
                RETURN;
            END_IF;
            IF NOT "P5001-DO" AND NOT (#"Comm-run"."in-timer".%X1 OR #"Comm-run"."in-timer".%X2) THEN
                "P5001-DO" := 1;
                #"Comm-run"."in-timer".%X1 := 1;
                #"Comm-run".step := 6;
                RETURN;
            END_IF;
            IF "P5001-DO" THEN
                #"Comm-run".step := 6;
            END_IF;
        END_IF;
        //step 6
        IF #"Comm-run".step = 6 THEN
            IF NOT "M5101-DO" AND (#"Comm-run"."in-timer".%X1 OR #"Comm-run"."in-timer".%X2)
                AND (#"Motor-Runtimer"[1].Q OR #"Motor-Runtimer"[2].Q) THEN
                "M5101-DO" := 1;
                #"Comm-run"."in-timer".%X1 := 0;
                #"Comm-run"."in-timer".%X2 := 1;
                #"Comm-run".step := 7;
                RETURN;
            END_IF;
            IF NOT "M5101-DO" AND NOT (#"Comm-run"."in-timer".%X1 OR #"Comm-run"."in-timer".%X2) THEN
                "M5101-DO" := 1;
                #"Comm-run"."in-timer".%X2 := 1;
                #"Comm-run".step := 7;
                RETURN;
            END_IF;
            IF "M5101-DO" THEN
                #"Comm-run".step := 7;
            END_IF;
        END_IF;
        //step 7
        IF #"Comm-run".step = 7 THEN
            IF NOT "P5008-DO" AND (#"Comm-run"."in-timer".%X1 OR #"Comm-run"."in-timer".%X2)
                AND (#"Motor-Runtimer"[1].Q OR #"Motor-Runtimer"[2].Q) THEN
                "P5008-DO" := 1;
                #"Comm-run"."in-timer".%X1 := 1;
                #"Comm-run"."in-timer".%X2 := 0;
                #"Comm-run".step := 8;
                RETURN;
            END_IF;
            IF NOT "P5008-DO" AND NOT (#"Comm-run"."in-timer".%X1 OR #"Comm-run"."in-timer".%X2) THEN
                "P5008-DO" := 1;
                #"Comm-run"."in-timer".%X1 := 1;
                #"Comm-run".step := 8;
                RETURN;
            END_IF;
            IF "P5008-DO" THEN
                #"Comm-run".step := 8;
            END_IF;
        END_IF;
        //step 8
        IF #"Comm-run".step = 8 THEN
            IF NOT "P5007-DO" AND (#"Comm-run"."in-timer".%X1 OR #"Comm-run"."in-timer".%X2)
                AND (#"Motor-Runtimer"[1].Q OR #"Motor-Runtimer"[2].Q) THEN
                "P5007-DO" := 1;
                #"Comm-run"."in-timer".%X1 := 0;
                #"Comm-run"."in-timer".%X2 := 1;
                #"Comm-run".step := 9;
                RETURN;
            END_IF;
            IF NOT "P5007-DO" AND NOT (#"Comm-run"."in-timer".%X1 OR #"Comm-run"."in-timer".%X2) THEN
                "P5007-DO" := 1;
                #"Comm-run"."in-timer".%X2 := 1;
                #"Comm-run".step := 9;
                RETURN;
            END_IF;
            IF "P5007-DO" THEN
                #"Comm-run".step := 9;
            END_IF;
        END_IF;
        //step 9
        IF #"Comm-run".step = 9 THEN
            IF NOT "M5004-DO" AND (#"Comm-run"."in-timer".%X1 OR #"Comm-run"."in-timer".%X2)
                AND (#"Motor-Runtimer"[1].Q OR #"Motor-Runtimer"[2].Q) THEN
                "M5004-DO" := 1;
                #"Comm-run"."in-timer".%X1 := 1;
                #"Comm-run"."in-timer".%X2 := 0;
                #"Comm-run".step := 10;
                RETURN;
            END_IF;
            IF NOT "M5004-DO" AND NOT (#"Comm-run"."in-timer".%X1 OR #"Comm-run"."in-timer".%X2) THEN
                "M5004-DO" := 1;
                #"Comm-run"."in-timer".%X1 := 1;
                #"Comm-run".step := 10;
                RETURN;
            END_IF;
            IF "M5004-DO" THEN
                #"Comm-run".step := 10;
            END_IF;
        END_IF;
        //step 10
        IF #"Comm-run".step = 10 THEN
            IF NOT "P5006-DO" AND (#"Comm-run"."in-timer".%X1 OR #"Comm-run"."in-timer".%X2)
                AND (#"Motor-Runtimer"[1].Q OR #"Motor-Runtimer"[2].Q) THEN
                "P5006-DO" := 1;
                #"Comm-run"."in-timer".%X1 := 0;
                #"Comm-run"."in-timer".%X2 := 1;
                #"Comm-run".step := 11;
                RETURN;
            END_IF;
            IF NOT "P5006-DO" AND NOT (#"Comm-run"."in-timer".%X1 OR #"Comm-run"."in-timer".%X2) THEN
                "P5006-DO" := 1;
                #"Comm-run"."in-timer".%X2 := 1;
                #"Comm-run".step := 11;
                RETURN;
            END_IF;
            IF "P5006-DO" THEN
                #"Comm-run".step := 11;
            END_IF;
        END_IF;
        //step 11
        IF #"Comm-run".step = 11 THEN
            IF NOT "P5005-DO" AND (#"Comm-run"."in-timer".%X1 OR #"Comm-run"."in-timer".%X2)
                AND (#"Motor-Runtimer"[1].Q OR #"Motor-Runtimer"[2].Q) THEN
                "P5005-DO" := 1;
                #"Comm-run"."in-timer".%X1 := 1;
                #"Comm-run"."in-timer".%X2 := 0;
                #"Comm-run".step := 12;
                RETURN;
            END_IF;
            IF NOT "P5005-DO" AND NOT (#"Comm-run"."in-timer".%X1 OR #"Comm-run"."in-timer".%X2) THEN
                "P5005-DO" := 1;
                #"Comm-run"."in-timer".%X1 := 1;
                #"Comm-run".step := 12;
                RETURN;
            END_IF;
            IF "P5005-DO" THEN
                #"Comm-run".step := 12;
            END_IF;
        END_IF;
        //step 12
        IF #"Comm-run".step = 12 THEN
            IF NOT "M5003-DO" AND (#"Comm-run"."in-timer".%X1 OR #"Comm-run"."in-timer".%X2)
                AND (#"Motor-Runtimer"[1].Q OR #"Motor-Runtimer"[2].Q) THEN
                "M5003-DO" := 1;
                #"Comm-run"."in-timer".%X1 := 0;
                #"Comm-run"."in-timer".%X2 := 1;
                #"Comm-run".step := 13;
                RETURN;
            END_IF;
            IF NOT "M5003-DO" AND NOT (#"Comm-run"."in-timer".%X1 OR #"Comm-run"."in-timer".%X2) THEN
                "M5003-DO" := 1;
                #"Comm-run"."in-timer".%X2 := 1;
                #"Comm-run".step := 13;
                RETURN;
            END_IF;
            IF "M5003-DO" THEN
                #"Comm-run".step := 13;
            END_IF;
        END_IF;
        //step 13
        IF #"Comm-run".step = 13 THEN
            IF NOT "P5004-DO" AND (#"Comm-run"."in-timer".%X1 OR #"Comm-run"."in-timer".%X2)
                AND (#"Motor-Runtimer"[1].Q OR #"Motor-Runtimer"[2].Q) THEN
                "P5004-DO" := 1;
                #"Comm-run"."in-timer".%X1 := 1;
                #"Comm-run"."in-timer".%X2 := 0;
                #"Comm-run".step := 14;
                RETURN;
            END_IF;
            IF NOT "P5004-DO" AND NOT (#"Comm-run"."in-timer".%X1 OR #"Comm-run"."in-timer".%X2) THEN
                "P5004-DO" := 1;
                #"Comm-run"."in-timer".%X1 := 1;
                #"Comm-run".step := 14;
                RETURN;
            END_IF;
            IF "P5004-DO" THEN
                #"Comm-run".step := 14;
            END_IF;
        END_IF;
        //step 14
        IF #"Comm-run".step = 14 THEN
            IF NOT "P5003-DO" AND (#"Comm-run"."in-timer".%X1 OR #"Comm-run"."in-timer".%X2)
                AND (#"Motor-Runtimer"[1].Q OR #"Motor-Runtimer"[2].Q) THEN
                "P5003-DO" := 1;
                #"Comm-run"."in-timer".%X1 := 0;
                #"Comm-run"."in-timer".%X2 := 1;
                #"Comm-run".step := 15;
                RETURN;
            END_IF;
            IF NOT "P5003-DO" AND NOT (#"Comm-run"."in-timer".%X1 OR #"Comm-run"."in-timer".%X2) THEN
                "P5003-DO" := 1;
                #"Comm-run"."in-timer".%X2 := 1;
                #"Comm-run".step := 15;
                RETURN;
            END_IF;
            IF "P5003-DO" THEN
                #"Comm-run".step := 15;
            END_IF;
        END_IF;
        //step 15
        IF #"Comm-run".step = 15 THEN
            IF NOT "M5002-DO" AND (#"Comm-run"."in-timer".%X1 OR #"Comm-run"."in-timer".%X2)
                AND (#"Motor-Runtimer"[1].Q OR #"Motor-Runtimer"[2].Q) THEN
                "M5002-DO" := 1;
                #"Comm-run".step := 16;
                RETURN;
            END_IF;
            IF NOT "M5002-DO" AND NOT (#"Comm-run"."in-timer".%X1 OR #"Comm-run"."in-timer".%X2) THEN
                "M5002-DO" := 1;
                #"Comm-run".step := 16;
                RETURN;
            END_IF;
            IF "M5002-DO" THEN
                #"Comm-run".step := 16;
            END_IF;
        END_IF;
        //step 16
        IF #"Comm-run".step = 16 THEN
            #"Comm-run"."in-timer" := 0;
            #"Comm-run".todo := 0;
            #"Comm-run".busy := 0;
            #"Comm-run".done := 1;
        END_IF;

    END_IF;
END_REGION

(* ---- SecondsConvert.st ---- *)
/* 变量声明 */
VAR_INPUT
    IN: REAL;
END_VAR
VAR_OUTPUT
    OUT: TIME;
END_VAR
VAR_TEMP
    temp-time:DINT;
END_VAR
VAR CONSTANT
    uint:REAL:=1000.0;
END_VAR

/* 转换逻辑，STL汇编语言，例如:输入1.5,输出1500. */
PROGRAM SecondsConvert
    L     #IN
    L     #unit
    *R
    RND
    T     #"temp-time"
    CALL  T_CONV
        src_type:=DInt
        dest_type:=Time
        IN  :=#"temp-time"
        OUT :=#OUT
END_PROGRAM

(* ---- Valve-v0.1.st ---- *)
REGION 预处理
    #open_timer_1(IN:=#i_open.%X1,
                  PT:=#open_time);
    #open_timer_2(IN := #i_open.%X2,
                  PT := #open_time);
    #open_timer_3(IN := #i_open.%X3,
                  PT := #open_time);
    #open_timer_4(IN := #i_open.%X4,
                  PT := #open_time);
    #open_timer_5(IN := #i_open.%X5,
                  PT := #open_time);
    #open_timer_6(IN := #i_open.%X6,
                  PT := #open_time);

    #close_timer_1(IN := #i_close.%X1,
                   PT := #close_time);
    #close_timer_2(IN := #i_close.%X2,
                   PT := #close_time);
    #close_timer_3(IN := #i_close.%X3,
                   PT := #close_time);
    #close_timer_4(IN := #i_close.%X4,
                   PT := #close_time);
    #close_timer_5(IN := #i_close.%X5,
                   PT := #close_time);
    #close_timer_6(IN := #i_close.%X6,
                   PT := #close_time);
    #loop_timer(IN := #b_loop,
                PT := #loop_time);
    #"pre-run-timer"(IN := #busy,
                     PT := #"pre-run-time");

    IF NOT(#Mode=5) AND #Mode=1 THEN

        #busy := TRUE;
    ELSE
        #busy := FALSE;
        #out_open := 0;
        #out_close := 0;
        #i_open := 0;
        #i_close := 0;
        #i_step := 0;
    END_IF;

END_REGION

REGION 球阀循环控制

    IF #"pre-run-timer".Q THEN

        //1 step
        IF #i_step = 0 THEN
            #out_close := 0;

            IF #b_loop AND #loop_timer.Q THEN
                #i_open.%X5 := FALSE;
                #out_open.%X1 := TRUE;
                #i_open.%X1 := TRUE;
                #i_close.%X1 := TRUE;

                IF #close_timer_1.Q THEN
                    #out_open.%X1 := FALSE;
                    #out_close.%X1 := TRUE;
                    #i_close.%X1 := FALSE;
                    #i_step := 1;
                END_IF;
            END_IF;
            IF NOT #b_loop THEN

                #out_open.%X1 := TRUE;
                #i_open.%X1 := TRUE;
                #i_close.%X1 := TRUE;

                IF #close_timer_1.Q THEN
                    #out_open.%X1 := FALSE;
                    #out_close.%X1 := TRUE;
                    #i_close.%X1 := FALSE;
                    #i_step := 1;

                END_IF;

            END_IF;
        END_IF;

        //2 step
        IF #i_step=1 AND #i_open.%X1 AND #open_timer_1.Q THEN
                #i_open.%X6 := FALSE;
                #out_open.%X2 := TRUE;
                #i_open.%X2 := TRUE;
                #i_close.%X2 := TRUE;

                IF #close_timer_2.Q THEN
                    #out_open.%X2 := FALSE;
                    #out_close.%X2 := TRUE;
                    #i_close.%X2 := FALSE;
                    #i_step := 2;

                END_IF;

            END_IF;

            //3 step
            IF #i_step = 2 AND #i_open.%X2 AND #open_timer_2.Q THEN
                #i_open.%X1 := FALSE;
                #out_open.%X3 := TRUE;
                #i_open.%X3 := TRUE;
                #i_close.%X3 := TRUE;

                IF #close_timer_3.Q THEN
                    #out_open.%X3 := FALSE;
                    #out_close.%X3 := TRUE;
                    #i_close.%X3 := FALSE;
                    #i_step := 3;

                END_IF;

            END_IF;

            //4 step
            IF #i_step = 3 AND #i_open.%X3 AND #open_timer_3.Q THEN
                #i_open.%X2 := FALSE;
                #out_open.%X4 := TRUE;
                #i_open.%X4 := TRUE;
                #i_close.%X4 := TRUE;

                IF #close_timer_4.Q THEN
                    #out_open.%X4 := FALSE;
                    #out_close.%X4 := TRUE;
                    #i_close.%X4 := FALSE;
                    #i_step := 4;

                END_IF;

            END_IF;

            //5 step
            IF #i_step = 4 AND #i_open.%X4 AND #open_timer_4.Q THEN
                #i_open.%X3 := FALSE;
                #out_open.%X5 := TRUE;
                #i_open.%X5 := TRUE;
                #i_close.%X5 := TRUE;

                IF #close_timer_5.Q THEN
                    #out_open.%X5 := FALSE;
                    #out_close.%X5 := TRUE;
                    #i_close.%X5 := FALSE;
                    #i_step := 5;

                END_IF;

            END_IF;

            //6 step
            IF #i_step = 5 AND #i_open.%X5 AND #open_timer_5.Q THEN
                #b_loop := 0;
                #i_open.%X4 := FALSE;
                #out_open.%X6 := TRUE;

                #i_close.%X6 := TRUE;

                IF #close_timer_6.Q THEN
                    #out_open.%X6 := FALSE;
                    #out_close.%X6 := TRUE;
                    #b_loop := 1;
                    #i_close.%X6 := FALSE;
                    #i_step := 0;
                END_IF;

            END_IF;

    END_IF;

END_REGION
